LIN {X -0.182,Y -626.109,Z 300.159,A 0.000,B 0.000,C 90.000,E1 244.717} C_DIS
LIN {X -0.135,Y -624.501,Z 300.155,A 0.000,B 0.000,C 90.000,E1 243.948} C_DIS
LIN {X -0.103,Y -622.641,Z 300.151,A 0.000,B 0.000,C 90.000,E1 243.179} C_DIS
LIN {X -0.091,Y -619.995,Z 300.145,A 0.000,B 0.000,C 90.000,E1 242.153} C_DIS
LIN {X 0.159,Y -616.323,Z 300.138,A 0.000,B 0.000,C 90.000,E1 240.845} C_DIS
LIN {X -0.188,Y -612.551,Z 300.131,A 0.000,B 0.000,C 90.000,E1 239.587} C_DIS
LIN {X -0.081,Y -608.634,Z 300.124,A 0.000,B 0.000,C 90.000,E1 238.280} C_DIS
LIN {X 0.080,Y -604.709,Z 300.117,A 0.000,B 0.000,C 90.000,E1 236.962} C_DIS
LIN {X 0.094,Y -599.962,Z 300.108,A 0.000,B 0.000,C 90.000,E1 235.388} C_DIS
LIN {X -0.124,Y -596.687,Z 300.102,A 0.000,B 0.000,C 90.000,E1 234.356} C_DIS
LIN {X -0.079,Y -591.376,Z 300.093,A 0.000,B 0.000,C 90.000,E1 232.763} C_DIS
LIN {X -0.207,Y -584.502,Z 300.081,A 0.000,B 0.000,C 90.000,E1 230.642} C_DIS
LIN {X -0.209,Y -580.122,Z 300.074,A 0.000,B 0.000,C 90.000,E1 229.299} C_DIS
LIN {X 0.078,Y -573.427,Z 300.062,A 0.000,B 0.000,C 90.000,E1 227.106} C_DIS
LIN {X 0.222,Y -569.220,Z 300.054,A 0.000,B 0.000,C 90.000,E1 225.729} C_DIS
LIN {X -0.015,Y -564.128,Z 300.045,A 0.000,B 0.000,C 90.000,E1 224.109} C_DIS
LIN {X -0.037,Y -559.947,Z 300.037,A 0.000,B 0.000,C 90.000,E1 222.732} C_DIS
LIN {X -0.107,Y -555.813,Z 300.030,A 0.000,B 0.000,C 90.000,E1 221.353} C_DIS
LIN {X 0.230,Y -550.744,Z 300.020,A 0.000,B 0.000,C 90.000,E1 219.644} C_DIS
LIN {X -0.267,Y -544.758,Z 300.009,A 0.000,B 0.000,C 90.000,E1 217.729} C_DIS
LIN {X -0.126,Y -541.410,Z 300.003,A 0.000,B 0.000,C 90.000,E1 216.583} C_DIS
LIN {X 0.135,Y -534.785,Z 299.991,A 0.000,B 0.000,C 90.000,E1 214.278} C_DIS
LIN {X -0.097,Y -528.365,Z 299.978,A 0.000,B 0.000,C 90.000,E1 212.005} C_DIS
LIN {X -0.297,Y -523.035,Z 299.967,A 0.000,B 0.000,C 90.000,E1 210.001} C_DIS
LIN {X 0.222,Y -519.344,Z 299.958,A 0.000,B 0.000,C 90.000,E1 208.487} C_DIS
LIN {X -0.257,Y -514.359,Z 299.947,A 0.000,B 0.000,C 90.000,E1 206.488} C_DIS
LIN {X 0.058,Y -509.624,Z 299.936,A 0.000,B 0.000,C 90.000,E1 204.387} C_DIS
LIN {X -0.170,Y -505.196,Z 299.924,A 0.000,B 0.000,C 90.000,E1 202.333} C_DIS
LIN {X -0.150,Y -500.375,Z 299.911,A 0.000,B 0.000,C 90.000,E1 199.939} C_DIS
LIN {X -0.081,Y -495.359,Z 299.896,A 0.000,B 0.000,C 90.000,E1 197.221} C_DIS
LIN {X 0.007,Y -490.770,Z 299.880,A 0.000,B 0.000,C 90.000,E1 194.481} C_DIS
LIN {X 0.162,Y -488.457,Z 299.872,A 0.000,B 0.000,C 90.000,E1 192.939} C_DIS
LIN {X 0.166,Y -484.922,Z 299.858,A 0.000,B 0.000,C 90.000,E1 190.489} C_DIS
LIN {X -0.009,Y -481.708,Z 299.845,A 0.000,B 0.000,C 90.000,E1 188.049} C_DIS
LIN {X -0.052,Y -479.486,Z 299.834,A 0.000,B 0.000,C 90.000,E1 186.201} C_DIS
LIN {X -0.099,Y -476.814,Z 299.821,A 0.000,B 0.000,C 90.000,E1 183.726} C_DIS
LIN {X -0.082,Y -474.710,Z 299.809,A 0.000,B 0.000,C 90.000,E1 181.547} C_DIS
LIN {X 0.154,Y -472.452,Z 299.791,A 0.000,B 0.000,C 90.000,E1 178.396} C_DIS
LIN {X -0.120,Y -470.977,Z 299.774,A 0.000,B 0.000,C 90.000,E1 175.298} C_DIS
LIN {X -0.174,Y -470.415,Z 299.762,A 0.000,B 0.000,C 90.000,E1 173.109} C_DIS
LIN {X -0.218,Y -470.146,Z 299.753,A 0.000,B 0.000,C 90.000,E1 171.546} C_DIS
LIN {X -0.165,Y -470.044,Z 299.741,A 0.000,B 0.000,C 90.000,E1 169.342} C_DIS
LIN {X -0.162,Y -470.689,Z 299.720,A 0.000,B 0.000,C 90.000,E1 165.574} C_DIS
LIN {X 0.121,Y -471.798,Z 299.706,A 0.000,B 0.000,C 90.000,E1 163.032} C_DIS
LIN {X -0.060,Y -473.445,Z 299.692,A 0.000,B 0.000,C 90.000,E1 160.550} C_DIS
LIN {X 0.149,Y -475.397,Z 299.678,A 0.000,B 0.000,C 90.000,E1 158.028} C_DIS
LIN {X 0.148,Y -478.180,Z 299.663,A 0.000,B 0.000,C 90.000,E1 155.229} C_DIS
LIN {X 0.212,Y -481.326,Z 299.649,A 0.000,B 0.000,C 90.000,E1 152.743} C_DIS
LIN {X -0.264,Y -485.148,Z 299.635,A 0.000,B 0.000,C 90.000,E1 150.333} C_DIS
LIN {X -0.010,Y -487.281,Z 299.628,A 0.000,B 0.000,C 90.000,E1 149.076} C_DIS
LIN {X 0.181,Y -491.179,Z 299.616,A 0.000,B 0.000,C 90.000,E1 146.914} C_DIS
LIN {X 0.075,Y -494.680,Z 299.606,A 0.000,B 0.000,C 90.000,E1 145.102} C_DIS
LIN {X -0.221,Y -497.526,Z 299.598,A 0.000,B 0.000,C 90.000,E1 143.623} C_DIS
LIN {X -0.045,Y -499.723,Z 299.591,A 0.000,B 0.000,C 90.000,E1 142.396} C_DIS
LIN {X 0.044,Y -502.272,Z 299.583,A 0.000,B 0.000,C 90.000,E1 140.884} C_DIS
LIN {X 0.009,Y -503.703,Z 299.578,A 0.000,B 0.000,C 90.000,E1 139.989} C_DIS
LIN {X 0.206,Y -505.330,Z 299.571,A 0.000,B 0.000,C 90.000,E1 138.771} C_DIS
LIN {X -0.174,Y -506.358,Z 299.566,A 0.000,B 0.000,C 90.000,E1 137.919} C_DIS
LIN {X 0.174,Y -507.145,Z 299.561,A 0.000,B 0.000,C 90.000,E1 136.986} C_DIS
LIN {X -0.075,Y -507.587,Z 299.558,A 0.000,B 0.000,C 90.000,E1 136.419} C_DIS
LIN {X 0.284,Y -508.000,Z 299.553,A 0.000,B 0.000,C 90.000,E1 135.486} C_DIS
LIN {X -0.197,Y -508.143,Z 299.546,A 0.000,B 0.000,C 90.000,E1 134.352} C_DIS
LIN {X 0.037,Y -507.836,Z 299.540,A 0.000,B 0.000,C 90.000,E1 133.137} C_DIS
LIN {X 0.055,Y -507.294,Z 299.535,A 0.000,B 0.000,C 90.000,E1 132.243} C_DIS
LIN {X 0.031,Y -506.498,Z 299.530,A 0.000,B 0.000,C 90.000,E1 131.353} C_DIS
LIN {X 0.150,Y -504.769,Z 299.522,A 0.000,B 0.000,C 90.000,E1 129.850} C_DIS
LIN {X -0.197,Y -502.345,Z 299.512,A 0.000,B 0.000,C 90.000,E1 128.096} C_DIS
LIN {X 0.044,Y -500.568,Z 299.505,A 0.000,B 0.000,C 90.000,E1 126.870} C_DIS
LIN {X -0.039,Y -498.718,Z 299.498,A 0.000,B 0.000,C 90.000,E1 125.678} C_DIS
LIN {X -0.146,Y -496.550,Z 299.492,A 0.000,B 0.000,C 90.000,E1 124.485} C_DIS
LIN {X -0.021,Y -493.751,Z 299.483,A 0.000,B 0.000,C 90.000,E1 122.959} C_DIS
LIN {X -0.222,Y -490.785,Z 299.475,A 0.000,B 0.000,C 90.000,E1 121.465} C_DIS
LIN {X -0.066,Y -487.195,Z 299.465,A 0.000,B 0.000,C 90.000,E1 119.617} C_DIS
LIN {X 0.211,Y -484.805,Z 299.458,A 0.000,B 0.000,C 90.000,E1 118.359} C_DIS
LIN {X -0.021,Y -480.543,Z 299.446,A 0.000,B 0.000,C 90.000,E1 116.232} C_DIS
LIN {X -0.144,Y -476.269,Z 299.434,A 0.000,B 0.000,C 90.000,E1 114.079} C_DIS
LIN {X -0.141,Y -472.067,Z 299.422,A 0.000,B 0.000,C 90.000,E1 111.897} C_DIS
LIN {X -0.207,Y -467.442,Z 299.408,A 0.000,B 0.000,C 90.000,E1 109.396} C_DIS
LIN {X -0.204,Y -463.065,Z 299.394,A 0.000,B 0.000,C 90.000,E1 106.913} C_DIS
LIN {X 0.198,Y -463.061,Z 299.394,A 0.000,B 0.000,C 90.000,E1 106.858} C_DIS
LIN {X -0.082,Y -467.666,Z 299.383,A 0.000,B 0.000,C 90.000,E1 104.954} C_DIS
LIN {X -0.093,Y -473.980,Z 299.362,A 0.000,B 0.000,C 90.000,E1 101.186} C_DIS
LIN {X -0.125,Y -475.882,Z 299.357,A 0.000,B 0.000,C 90.000,E1 100.254} C_DIS
LIN {X 0.183,Y -476.341,Z 299.355,A 0.000,B 0.000,C 90.000,E1 99.905} C_DIS
LIN {X 0.140,Y -481.850,Z 299.331,A 0.000,B 0.000,C 90.000,E1 95.568} C_DIS
LIN {X -0.013,Y -482.187,Z 299.329,A 0.000,B 0.000,C 90.000,E1 95.277} C_DIS
LIN {X -0.079,Y -485.348,Z 299.305,A 0.000,B 0.000,C 90.000,E1 90.974} C_DIS
LIN {X 0.230,Y -485.533,Z 299.304,A 0.000,B 0.000,C 90.000,E1 90.630} C_DIS
LIN {X -0.047,Y -486.338,Z 299.282,A 0.000,B 0.000,C 90.000,E1 86.674} C_DIS
LIN {X 0.088,Y -486.278,Z 299.278,A 0.000,B 0.000,C 90.000,E1 86.045} C_DIS
LIN {X -0.193,Y -484.694,Z 299.254,A 0.000,B 0.000,C 90.000,E1 81.781} C_DIS
LIN {X 0.155,Y -484.553,Z 299.253,A 0.000,B 0.000,C 90.000,E1 81.432} C_DIS
LIN {X 0.024,Y -480.493,Z 299.227,A 0.000,B 0.000,C 90.000,E1 76.825} C_DIS
LIN {X 0.147,Y -474.643,Z 299.203,A 0.000,B 0.000,C 90.000,E1 72.543} C_DIS
LIN {X -0.098,Y -481.750,Z 299.187,A 0.000,B 0.000,C 90.000,E1 69.699} C_DIS
LIN {X -0.059,Y -487.505,Z 299.175,A 0.000,B 0.000,C 90.000,E1 67.539} C_DIS
LIN {X -0.122,Y -493.376,Z 299.163,A 0.000,B 0.000,C 90.000,E1 65.409} C_DIS
LIN {X 0.177,Y -499.347,Z 299.152,A 0.000,B 0.000,C 90.000,E1 63.256} C_DIS
LIN {X 0.100,Y -504.591,Z 299.142,A 0.000,B 0.000,C 90.000,E1 61.463} C_DIS
LIN {X -0.188,Y -510.675,Z 299.130,A 0.000,B 0.000,C 90.000,E1 59.410} C_DIS
LIN {X -0.053,Y -516.724,Z 299.118,A 0.000,B 0.000,C 90.000,E1 57.327} C_DIS
LIN {X -0.240,Y -520.932,Z 299.110,A 0.000,B 0.000,C 90.000,E1 55.881} C_DIS
LIN {X -0.012,Y -524.250,Z 299.104,A 0.000,B 0.000,C 90.000,E1 54.689} C_DIS
LIN {X 0.239,Y -528.043,Z 299.096,A 0.000,B 0.000,C 90.000,E1 53.210} C_DIS
LIN {X 0.166,Y -530.153,Z 299.091,A 0.000,B 0.000,C 90.000,E1 52.351} C_DIS
LIN {X -0.317,Y -532.828,Z 299.085,A 0.000,B 0.000,C 90.000,E1 51.251} C_DIS
LIN {X -0.017,Y -535.818,Z 299.077,A 0.000,B 0.000,C 90.000,E1 49.784} C_DIS
LIN {X -0.083,Y -537.922,Z 299.070,A 0.000,B 0.000,C 90.000,E1 48.647} C_DIS
LIN {X 0.243,Y -539.780,Z 299.064,A 0.000,B 0.000,C 90.000,E1 47.472} C_DIS
LIN {X 0.225,Y -540.990,Z 299.059,A 0.000,B 0.000,C 90.000,E1 46.620} C_DIS
LIN {X 0.210,Y -542.324,Z 299.053,A 0.000,B 0.000,C 90.000,E1 45.486} C_DIS
LIN {X -0.171,Y -543.078,Z 299.048,A 0.000,B 0.000,C 90.000,E1 44.676} C_DIS
LIN {X -0.157,Y -543.869,Z 299.042,A 0.000,B 0.000,C 90.000,E1 43.542} C_DIS
LIN {X -0.098,Y -544.655,Z 299.032,A 0.000,B 0.000,C 90.000,E1 41.838} C_DIS
LIN {X -0.032,Y -544.905,Z 299.026,A 0.000,B 0.000,C 90.000,E1 40.701} C_DIS
LIN {X 0.035,Y -544.893,Z 299.020,A 0.000,B 0.000,C 90.000,E1 39.564} C_DIS
LIN {X -0.282,Y -544.756,Z 299.015,A 0.000,B 0.000,C 90.000,E1 38.749} C_DIS
LIN {X -0.174,Y -544.378,Z 299.010,A 0.000,B 0.000,C 90.000,E1 37.890} C_DIS
LIN {X 0.005,Y -543.528,Z 299.003,A 0.000,B 0.000,C 90.000,E1 36.457} C_DIS
LIN {X 0.133,Y -542.653,Z 298.996,A 0.000,B 0.000,C 90.000,E1 35.311} C_DIS
LIN {X -0.044,Y -541.479,Z 298.988,A 0.000,B 0.000,C 90.000,E1 33.913} C_DIS
LIN {X 0.201,Y -540.148,Z 298.981,A 0.000,B 0.000,C 90.000,E1 32.467} C_DIS
LIN {X -0.148,Y -538.516,Z 298.971,A 0.000,B 0.000,C 90.000,E1 30.797} C_DIS
LIN {X -0.062,Y -536.827,Z 298.962,A 0.000,B 0.000,C 90.000,E1 29.077} C_DIS
LIN {X -0.080,Y -534.816,Z 298.950,A 0.000,B 0.000,C 90.000,E1 27.078} C_DIS
LIN {X -0.152,Y -532.853,Z 298.939,A 0.000,B 0.000,C 90.000,E1 25.079} C_DIS
LIN {X 0.131,Y -530.506,Z 298.925,A 0.000,B 0.000,C 90.000,E1 22.461} C_DIS
LIN {X 0.132,Y -528.251,Z 298.909,A 0.000,B 0.000,C 90.000,E1 19.577} C_DIS
LIN {X 0.020,Y -526.719,Z 298.896,A 0.000,B 0.000,C 90.000,E1 17.275} C_DIS
LIN {X 0.217,Y -525.316,Z 298.880,A 0.000,B 0.000,C 90.000,E1 14.356} C_DIS
LIN {X -0.064,Y -524.607,Z 298.869,A 0.000,B 0.000,C 90.000,E1 12.355} C_DIS
LIN {X 0.027,Y -524.180,Z 298.859,A 0.000,B 0.000,C 90.000,E1 10.602} C_DIS
LIN {X 0.028,Y -523.977,Z 298.848,A 0.000,B 0.000,C 90.000,E1 8.568} C_DIS
LIN {X -0.116,Y -524.085,Z 298.835,A 0.000,B 0.000,C 90.000,E1 6.258} C_DIS
LIN {X -0.217,Y -524.347,Z 298.827,A 0.000,B 0.000,C 90.000,E1 4.816} C_DIS
LIN {X 0.208,Y -524.558,Z 298.822,A 0.000,B 0.000,C 90.000,E1 3.898} C_DIS
LIN {X 0.074,Y -525.115,Z 298.815,A 0.000,B 0.000,C 90.000,E1 2.751} C_DIS
LIN {X -0.088,Y -525.738,Z 298.807,A 0.000,B 0.000,C 90.000,E1 1.318} C_DIS
LIN {X 0.015,Y -527.991,Z 298.788,A 0.000,B 0.000,C 90.000,E1 357.764} C_DIS
LIN {X -0.105,Y -529.771,Z 298.776,A 0.000,B 0.000,C 90.000,E1 355.755} C_DIS
LIN {X 0.151,Y -537.369,Z 298.744,A 0.000,B 0.000,C 90.000,E1 349.982} C_DIS
LIN {X 0.274,Y -546.360,Z 298.722,A 0.000,B 0.000,C 90.000,E1 345.992} C_DIS
LIN {X -0.070,Y -550.608,Z 298.713,A 0.000,B 0.000,C 90.000,E1 344.338} C_DIS
LIN {X 0.092,Y -555.900,Z 298.702,A 0.000,B 0.000,C 90.000,E1 342.362} C_DIS
LIN {X 0.033,Y -561.563,Z 298.691,A 0.000,B 0.000,C 90.000,E1 340.423} C_DIS
LIN {X -0.088,Y -568.480,Z 298.679,A 0.000,B 0.000,C 90.000,E1 338.230} C_DIS
LIN {X -0.154,Y -573.017,Z 298.671,A 0.000,B 0.000,C 90.000,E1 336.869} C_DIS
LIN {X -0.063,Y -578.480,Z 298.662,A 0.000,B 0.000,C 90.000,E1 335.229} C_DIS
LIN {X 0.019,Y -585.185,Z 298.652,A 0.000,B 0.000,C 90.000,E1 333.332} C_DIS
LIN {X 0.213,Y -589.950,Z 298.644,A 0.000,B 0.000,C 90.000,E1 331.975} C_DIS
LIN {X -0.028,Y -594.540,Z 298.637,A 0.000,B 0.000,C 90.000,E1 330.667} C_DIS
LIN {X 0.245,Y -600.852,Z 298.627,A 0.000,B 0.000,C 90.000,E1 328.791} C_DIS
LIN {X 0.368,Y -609.059,Z 298.614,A 0.000,B 0.000,C 90.000,E1 326.421} C_DIS
LIN {X -0.242,Y -616.568,Z 298.602,A 0.000,B 0.000,C 90.000,E1 324.402} C_DIS
LIN {X 0.137,Y -620.115,Z 298.596,A 0.000,B 0.000,C 90.000,E1 323.336} C_DIS
LIN {X 0.072,Y -623.435,Z 298.591,A 0.000,B 0.000,C 90.000,E1 322.316} C_DIS
LIN {X 0.003,Y -627.305,Z 298.584,A 0.000,B 0.000,C 90.000,E1 321.045} C_DIS
LIN {X -0.235,Y -631.904,Z 298.575,A 0.000,B 0.000,C 90.000,E1 319.542} C_DIS
LIN {X 0.147,Y -635.674,Z 298.568,A 0.000,B 0.000,C 90.000,E1 318.243} C_DIS
LIN {X 0.240,Y -642.093,Z 298.556,A 0.000,B 0.000,C 90.000,E1 315.972} C_DIS
LIN {X -0.207,Y -646.536,Z 298.547,A 0.000,B 0.000,C 90.000,E1 314.514} C_DIS
LIN {X -0.049,Y -649.984,Z 298.540,A 0.000,B 0.000,C 90.000,E1 313.257} C_DIS
LIN {X 0.170,Y -653.282,Z 298.533,A 0.000,B 0.000,C 90.000,E1 312.000} C_DIS
LIN {X 0.027,Y -655.124,Z 298.529,A 0.000,B 0.000,C 90.000,E1 311.272} C_DIS
LIN {X -0.082,Y -657.386,Z 298.524,A 0.000,B 0.000,C 90.000,E1 310.297} C_DIS
LIN {X 0.349,Y -659.514,Z 298.518,A 0.000,B 0.000,C 90.000,E1 309.277} C_DIS
LIN {X -0.147,Y -661.854,Z 298.512,A 0.000,B 0.000,C 90.000,E1 308.096} C_DIS
LIN {X 0.347,Y -663.452,Z 298.506,A 0.000,B 0.000,C 90.000,E1 307.076} C_DIS
LIN {X -0.030,Y -664.474,Z 298.502,A 0.000,B 0.000,C 90.000,E1 306.377} C_DIS
LIN {X -0.007,Y -665.299,Z 298.498,A 0.000,B 0.000,C 90.000,E1 305.644} C_DIS
LIN {X 0.061,Y -665.747,Z 298.495,A 0.000,B 0.000,C 90.000,E1 305.152} C_DIS
LIN {X 0.327,Y -666.190,Z 298.489,A 0.000,B 0.000,C 90.000,E1 303.913} C_DIS
LIN {X -0.026,Y -666.275,Z 298.485,A 0.000,B 0.000,C 90.000,E1 303.214} C_DIS
LIN {X 0.312,Y -665.993,Z 298.479,A 0.000,B 0.000,C 90.000,E1 302.212} C_DIS
LIN {X 0.026,Y -665.658,Z 298.476,A 0.000,B 0.000,C 90.000,E1 301.750} C_DIS
LIN {X 0.227,Y -664.792,Z 298.472,A 0.000,B 0.000,C 90.000,E1 301.003} C_DIS
LIN {X 0.078,Y -663.635,Z 298.468,A 0.000,B 0.000,C 90.000,E1 300.285} C_DIS
LIN {X -0.190,Y -661.626,Z 298.463,A 0.000,B 0.000,C 90.000,E1 299.333} C_DIS
LIN {X -0.236,Y -659.458,Z 298.457,A 0.000,B 0.000,C 90.000,E1 298.359} C_DIS
LIN {X -0.186,Y -656.523,Z 298.451,A 0.000,B 0.000,C 90.000,E1 297.129} C_DIS
LIN {X -0.192,Y -653.341,Z 298.444,A 0.000,B 0.000,C 90.000,E1 295.899} C_DIS
LIN {X -0.050,Y -650.744,Z 298.438,A 0.000,B 0.000,C 90.000,E1 294.899} C_DIS
LIN {X 0.156,Y -647.411,Z 298.431,A 0.000,B 0.000,C 90.000,E1 293.643} C_DIS
LIN {X 0.122,Y -643.343,Z 298.423,A 0.000,B 0.000,C 90.000,E1 292.153} C_DIS
LIN {X 0.003,Y -639.359,Z 298.415,A 0.000,B 0.000,C 90.000,E1 290.663} C_DIS
LIN {X 0.169,Y -635.540,Z 298.406,A 0.000,B 0.000,C 90.000,E1 289.141} C_DIS
LIN {X 0.083,Y -629.583,Z 298.392,A 0.000,B 0.000,C 90.000,E1 286.622} C_DIS
LIN {X 0.239,Y -624.337,Z 298.378,A 0.000,B 0.000,C 90.000,E1 284.064} C_DIS
LIN {X 0.299,Y -619.586,Z 298.363,A 0.000,B 0.000,C 90.000,E1 281.243} C_DIS
LIN {X -0.158,Y -616.056,Z 298.347,A 0.000,B 0.000,C 90.000,E1 278.454} C_DIS
LIN {X -0.290,Y -613.529,Z 298.331,A 0.000,B 0.000,C 90.000,E1 275.625} C_DIS
LIN {X -0.019,Y -612.132,Z 298.315,A 0.000,B 0.000,C 90.000,E1 272.751} C_DIS
LIN {X -0.136,Y -611.738,Z 298.304,A 0.000,B 0.000,C 90.000,E1 270.688} C_DIS
LIN {X -0.289,Y -612.009,Z 298.289,A 0.000,B 0.000,C 90.000,E1 268.108} C_DIS
LIN {X -0.093,Y -614.280,Z 298.268,A 0.000,B 0.000,C 90.000,E1 264.204} C_DIS
LIN {X -0.260,Y -616.461,Z 298.255,A 0.000,B 0.000,C 90.000,E1 261.894} C_DIS
LIN {X -0.129,Y -620.046,Z 298.239,A 0.000,B 0.000,C 90.000,E1 259.050} C_DIS
LIN {X -0.073,Y -623.099,Z 298.228,A 0.000,B 0.000,C 90.000,E1 256.992} C_DIS
LIN {X 0.084,Y -625.017,Z 298.221,A 0.000,B 0.000,C 90.000,E1 255.700} C_DIS
LIN {X 0.024,Y -626.507,Z 298.215,A 0.000,B 0.000,C 90.000,E1 254.685} C_DIS
LIN {X 0.018,Y -627.423,Z 298.211,A 0.000,B 0.000,C 90.000,E1 253.921} C_DIS
LIN {X -0.011,Y -628.337,Z 298.205,A 0.000,B 0.000,C 90.000,E1 252.906} C_DIS
LIN {X -0.241,Y -629.516,Z 298.197,A 0.000,B 0.000,C 90.000,E1 251.402} C_DIS
LIN {X 0.155,Y -629.873,Z 298.192,A 0.000,B 0.000,C 90.000,E1 250.604} C_DIS
LIN {X 0.355,Y -630.024,Z 298.187,A 0.000,B 0.000,C 90.000,E1 249.571} C_DIS
LIN {X -0.037,Y -629.773,Z 298.181,A 0.000,B 0.000,C 90.000,E1 248.592} C_DIS
LIN {X -0.236,Y -629.487,Z 298.178,A 0.000,B 0.000,C 90.000,E1 248.103} C_DIS
LIN {X 0.179,Y -628.629,Z 298.173,A 0.000,B 0.000,C 90.000,E1 247.050} C_DIS
LIN {X -0.015,Y -627.694,Z 298.168,A 0.000,B 0.000,C 90.000,E1 246.305} C_DIS
LIN {X -0.195,Y -625.621,Z 298.161,A 0.000,B 0.000,C 90.000,E1 245.049} C_DIS
LIN {X -0.159,Y -624.119,Z 298.157,A 0.000,B 0.000,C 90.000,E1 244.280} C_DIS
LIN {X -0.135,Y -622.359,Z 298.153,A 0.000,B 0.000,C 90.000,E1 243.512} C_DIS
LIN {X -0.136,Y -619.093,Z 298.146,A 0.000,B 0.000,C 90.000,E1 242.231} C_DIS
LIN {X 0.093,Y -615.474,Z 298.139,A 0.000,B 0.000,C 90.000,E1 240.923} C_DIS
LIN {X -0.272,Y -611.743,Z 298.131,A 0.000,B 0.000,C 90.000,E1 239.665} C_DIS
LIN {X 0.137,Y -607.865,Z 298.124,A 0.000,B 0.000,C 90.000,E1 238.329} C_DIS
LIN {X -0.039,Y -603.959,Z 298.117,A 0.000,B 0.000,C 90.000,E1 237.041} C_DIS
LIN {X 0.051,Y -599.975,Z 298.110,A 0.000,B 0.000,C 90.000,E1 235.722} C_DIS
LIN {X -0.160,Y -596.694,Z 298.104,A 0.000,B 0.000,C 90.000,E1 234.689} C_DIS
LIN {X -0.074,Y -593.204,Z 298.098,A 0.000,B 0.000,C 90.000,E1 233.623} C_DIS
LIN {X 0.111,Y -587.118,Z 298.088,A 0.000,B 0.000,C 90.000,E1 231.743} C_DIS
LIN {X -0.217,Y -582.880,Z 298.080,A 0.000,B 0.000,C 90.000,E1 230.436} C_DIS
LIN {X 0.153,Y -575.978,Z 298.068,A 0.000,B 0.000,C 90.000,E1 228.243} C_DIS
LIN {X 0.073,Y -571.039,Z 298.059,A 0.000,B 0.000,C 90.000,E1 226.620} C_DIS
LIN {X -0.129,Y -565.920,Z 298.050,A 0.000,B 0.000,C 90.000,E1 225.000} C_DIS
LIN {X -0.026,Y -560.892,Z 298.041,A 0.000,B 0.000,C 90.000,E1 223.338} C_DIS
LIN {X -0.034,Y -555.877,Z 298.032,A 0.000,B 0.000,C 90.000,E1 221.676} C_DIS
LIN {X -0.113,Y -550.777,Z 298.022,A 0.000,B 0.000,C 90.000,E1 220.011} C_DIS
LIN {X 0.073,Y -546.500,Z 298.014,A 0.000,B 0.000,C 90.000,E1 218.588} C_DIS
LIN {X 0.298,Y -541.470,Z 298.005,A 0.000,B 0.000,C 90.000,E1 216.870} C_DIS
LIN {X 0.115,Y -534.747,Z 297.992,A 0.000,B 0.000,C 90.000,E1 214.612} C_DIS
LIN {X 0.296,Y -527.505,Z 297.978,A 0.000,B 0.000,C 90.000,E1 212.005} C_DIS
LIN {X -0.326,Y -522.900,Z 297.968,A 0.000,B 0.000,C 90.000,E1 210.335} C_DIS
LIN {X 0.237,Y -517.730,Z 297.957,A 0.000,B 0.000,C 90.000,E1 208.231} C_DIS
LIN {X -0.280,Y -512.769,Z 297.946,A 0.000,B 0.000,C 90.000,E1 206.232} C_DIS
LIN {X -0.321,Y -508.749,Z 297.936,A 0.000,B 0.000,C 90.000,E1 204.463} C_DIS
LIN {X 0.101,Y -504.343,Z 297.924,A 0.000,B 0.000,C 90.000,E1 202.333} C_DIS
LIN {X 0.093,Y -499.541,Z 297.911,A 0.000,B 0.000,C 90.000,E1 199.939} C_DIS
LIN {X 0.131,Y -494.572,Z 297.896,A 0.000,B 0.000,C 90.000,E1 197.221} C_DIS
LIN {X 0.192,Y -490.013,Z 297.881,A 0.000,B 0.000,C 90.000,E1 194.481} C_DIS
LIN {X -0.252,Y -487.727,Z 297.872,A 0.000,B 0.000,C 90.000,E1 193.008} C_DIS
LIN {X -0.163,Y -484.250,Z 297.859,A 0.000,B 0.000,C 90.000,E1 190.546} C_DIS
LIN {X 0.118,Y -481.096,Z 297.845,A 0.000,B 0.000,C 90.000,E1 188.049} C_DIS
LIN {X -0.097,Y -478.583,Z 297.833,A 0.000,B 0.000,C 90.000,E1 185.910} C_DIS
LIN {X -0.210,Y -476.033,Z 297.819,A 0.000,B 0.000,C 90.000,E1 183.440} C_DIS
LIN {X -0.210,Y -473.997,Z 297.807,A 0.000,B 0.000,C 90.000,E1 181.260} C_DIS
LIN {X -0.033,Y -472.274,Z 297.793,A 0.000,B 0.000,C 90.000,E1 178.740} C_DIS
LIN {X 0.162,Y -470.725,Z 297.776,A 0.000,B 0.000,C 90.000,E1 175.584} C_DIS
LIN {X -0.130,Y -470.076,Z 297.762,A 0.000,B 0.000,C 90.000,E1 173.109} C_DIS
LIN {X 0.001,Y -469.874,Z 297.755,A 0.000,B 0.000,C 90.000,E1 171.837} C_DIS
LIN {X -0.137,Y -469.675,Z 297.741,A 0.000,B 0.000,C 90.000,E1 169.342} C_DIS
LIN {X -0.085,Y -470.203,Z 297.722,A 0.000,B 0.000,C 90.000,E1 165.880} C_DIS
LIN {X -0.145,Y -471.236,Z 297.708,A 0.000,B 0.000,C 90.000,E1 163.378} C_DIS
LIN {X -0.035,Y -472.778,Z 297.694,A 0.000,B 0.000,C 90.000,E1 160.859} C_DIS
LIN {X 0.237,Y -473.976,Z 297.685,A 0.000,B 0.000,C 90.000,E1 159.263} C_DIS
LIN {X 0.024,Y -476.139,Z 297.671,A 0.000,B 0.000,C 90.000,E1 156.794} C_DIS
LIN {X -0.199,Y -479.259,Z 297.656,A 0.000,B 0.000,C 90.000,E1 154.024} C_DIS
LIN {X 0.106,Y -484.121,Z 297.637,A 0.000,B 0.000,C 90.000,E1 150.589} C_DIS
LIN {X -0.087,Y -486.691,Z 297.628,A 0.000,B 0.000,C 90.000,E1 149.076} C_DIS
LIN {X 0.088,Y -490.536,Z 297.616,A 0.000,B 0.000,C 90.000,E1 146.914} C_DIS
LIN {X 0.117,Y -493.407,Z 297.608,A 0.000,B 0.000,C 90.000,E1 145.388} C_DIS
LIN {X -0.205,Y -496.206,Z 297.599,A 0.000,B 0.000,C 90.000,E1 143.909} C_DIS
LIN {X -0.049,Y -498.408,Z 297.593,A 0.000,B 0.000,C 90.000,E1 142.683} C_DIS
LIN {X 0.017,Y -500.971,Z 297.584,A 0.000,B 0.000,C 90.000,E1 141.170} C_DIS
LIN {X -0.151,Y -502.860,Z 297.578,A 0.000,B 0.000,C 90.000,E1 139.989} C_DIS
LIN {X 0.033,Y -504.484,Z 297.571,A 0.000,B 0.000,C 90.000,E1 138.771} C_DIS
LIN {X 0.136,Y -505.242,Z 297.568,A 0.000,B 0.000,C 90.000,E1 138.162} C_DIS
LIN {X -0.247,Y -506.101,Z 297.563,A 0.000,B 0.000,C 90.000,E1 137.310} C_DIS
LIN {X 0.094,Y -506.767,Z 297.558,A 0.000,B 0.000,C 90.000,E1 136.377} C_DIS
LIN {X 0.077,Y -507.162,Z 297.553,A 0.000,B 0.000,C 90.000,E1 135.486} C_DIS
LIN {X 0.301,Y -507.308,Z 297.546,A 0.000,B 0.000,C 90.000,E1 134.271} C_DIS
LIN {X -0.061,Y -507.139,Z 297.541,A 0.000,B 0.000,C 90.000,E1 133.419} C_DIS
LIN {X 0.153,Y -506.426,Z 297.535,A 0.000,B 0.000,C 90.000,E1 132.204} C_DIS
LIN {X 0.160,Y -505.647,Z 297.530,A 0.000,B 0.000,C 90.000,E1 131.310} C_DIS
LIN {X -0.219,Y -504.645,Z 297.525,A 0.000,B 0.000,C 90.000,E1 130.458} C_DIS
LIN {X -0.020,Y -503.134,Z 297.518,A 0.000,B 0.000,C 90.000,E1 129.241} C_DIS
LIN {X 0.108,Y -501.090,Z 297.510,A 0.000,B 0.000,C 90.000,E1 127.729} C_DIS
LIN {X 0.075,Y -498.355,Z 297.500,A 0.000,B 0.000,C 90.000,E1 125.931} C_DIS
LIN {X 0.089,Y -496.811,Z 297.495,A 0.000,B 0.000,C 90.000,E1 125.025} C_DIS
LIN {X 0.066,Y -493.432,Z 297.485,A 0.000,B 0.000,C 90.000,E1 123.214} C_DIS
LIN {X 0.014,Y -491.122,Z 297.478,A 0.000,B 0.000,C 90.000,E1 122.005} C_DIS
LIN {X 0.178,Y -488.142,Z 297.469,A 0.000,B 0.000,C 90.000,E1 120.463} C_DIS
LIN {X 0.040,Y -485.166,Z 297.461,A 0.000,B 0.000,C 90.000,E1 118.949} C_DIS
LIN {X 0.052,Y -482.748,Z 297.454,A 0.000,B 0.000,C 90.000,E1 117.719} C_DIS
LIN {X 0.216,Y -479.099,Z 297.444,A 0.000,B 0.000,C 90.000,E1 115.848} C_DIS
LIN {X -0.119,Y -475.443,Z 297.433,A 0.000,B 0.000,C 90.000,E1 114.027} C_DIS
LIN {X -0.132,Y -471.269,Z 297.421,A 0.000,B 0.000,C 90.000,E1 111.844} C_DIS
LIN {X -0.059,Y -466.674,Z 297.407,A 0.000,B 0.000,C 90.000,E1 109.322} C_DIS
LIN {X 0.031,Y -462.724,Z 297.395,A 0.000,B 0.000,C 90.000,E1 107.040} C_DIS
LIN {X -0.010,Y -462.719,Z 297.395,A 0.000,B 0.000,C 90.000,E1 107.040} C_DIS
LIN {X -0.099,Y -467.796,Z 297.383,A 0.000,B 0.000,C 90.000,E1 104.898} C_DIS
LIN {X -0.128,Y -476.002,Z 297.357,A 0.000,B 0.000,C 90.000,E1 100.197} C_DIS
LIN {X -0.137,Y -477.010,Z 297.351,A 0.000,B 0.000,C 90.000,E1 99.265} C_DIS
LIN {X 0.146,Y -481.941,Z 297.331,A 0.000,B 0.000,C 90.000,E1 95.511} C_DIS
LIN {X -0.007,Y -482.210,Z 297.329,A 0.000,B 0.000,C 90.000,E1 95.220} C_DIS
LIN {X -0.068,Y -485.408,Z 297.305,A 0.000,B 0.000,C 90.000,E1 90.917} C_DIS
LIN {X 0.242,Y -485.528,Z 297.303,A 0.000,B 0.000,C 90.000,E1 90.573} C_DIS
LIN {X -0.036,Y -486.367,Z 297.281,A 0.000,B 0.000,C 90.000,E1 86.617} C_DIS
LIN {X -0.210,Y -486.367,Z 297.280,A 0.000,B 0.000,C 90.000,E1 86.331} C_DIS
LIN {X 0.124,Y -485.673,Z 297.273,A 0.000,B 0.000,C 90.000,E1 85.065} C_DIS
LIN {X -0.188,Y -484.691,Z 297.254,A 0.000,B 0.000,C 90.000,E1 81.724} C_DIS
LIN {X 0.160,Y -484.485,Z 297.252,A 0.000,B 0.000,C 90.000,E1 81.376} C_DIS
LIN {X 0.163,Y -480.661,Z 297.228,A 0.000,B 0.000,C 90.000,E1 77.061} C_DIS
LIN {X 0.129,Y -480.411,Z 297.227,A 0.000,B 0.000,C 90.000,E1 76.756} C_DIS
LIN {X -0.113,Y -474.423,Z 297.202,A 0.000,B 0.000,C 90.000,E1 72.362} C_DIS
LIN {X 0.048,Y -479.524,Z 297.190,A 0.000,B 0.000,C 90.000,E1 70.242} C_DIS
LIN {X -0.145,Y -485.198,Z 297.178,A 0.000,B 0.000,C 90.000,E1 68.103} C_DIS
LIN {X 0.123,Y -489.376,Z 297.170,A 0.000,B 0.000,C 90.000,E1 66.538} C_DIS
LIN {X -0.178,Y -493.591,Z 297.161,A 0.000,B 0.000,C 90.000,E1 65.049} C_DIS
LIN {X 0.013,Y -497.858,Z 297.153,A 0.000,B 0.000,C 90.000,E1 63.512} C_DIS
LIN {X 0.202,Y -503.972,Z 297.141,A 0.000,B 0.000,C 90.000,E1 61.385} C_DIS
LIN {X -0.092,Y -510.039,Z 297.130,A 0.000,B 0.000,C 90.000,E1 59.331} C_DIS
LIN {X -0.237,Y -514.395,Z 297.121,A 0.000,B 0.000,C 90.000,E1 57.867} C_DIS
LIN {X -0.035,Y -518.670,Z 297.113,A 0.000,B 0.000,C 90.000,E1 56.373} C_DIS
LIN {X 0.108,Y -522.812,Z 297.105,A 0.000,B 0.000,C 90.000,E1 54.895} C_DIS
LIN {X -0.088,Y -526.680,Z 297.097,A 0.000,B 0.000,C 90.000,E1 53.463} C_DIS
LIN {X 0.226,Y -529.520,Z 297.091,A 0.000,B 0.000,C 90.000,E1 52.271} C_DIS
LIN {X -0.264,Y -532.181,Z 297.084,A 0.000,B 0.000,C 90.000,E1 51.170} C_DIS
LIN {X 0.032,Y -534.577,Z 297.078,A 0.000,B 0.000,C 90.000,E1 49.989} C_DIS
LIN {X -0.046,Y -536.758,Z 297.071,A 0.000,B 0.000,C 90.000,E1 48.852} C_DIS
LIN {X -0.095,Y -538.647,Z 297.065,A 0.000,B 0.000,C 90.000,E1 47.715} C_DIS
LIN {X -0.125,Y -539.901,Z 297.060,A 0.000,B 0.000,C 90.000,E1 46.863} C_DIS
LIN {X -0.160,Y -541.317,Z 297.054,A 0.000,B 0.000,C 90.000,E1 45.729} C_DIS
LIN {X -0.169,Y -542.321,Z 297.048,A 0.000,B 0.000,C 90.000,E1 44.595} C_DIS
LIN {X -0.166,Y -543.093,Z 297.041,A 0.000,B 0.000,C 90.000,E1 43.461} C_DIS
LIN {X -0.125,Y -543.879,Z 297.032,A 0.000,B 0.000,C 90.000,E1 41.757} C_DIS
LIN {X -0.072,Y -544.051,Z 297.026,A 0.000,B 0.000,C 90.000,E1 40.620} C_DIS
LIN {X -0.049,Y -544.039,Z 297.021,A 0.000,B 0.000,C 90.000,E1 39.769} C_DIS
LIN {X 0.045,Y -543.894,Z 297.016,A 0.000,B 0.000,C 90.000,E1 38.910} C_DIS
LIN {X -0.282,Y -543.593,Z 297.012,A 0.000,B 0.000,C 90.000,E1 38.096} C_DIS
LIN {X -0.120,Y -542.787,Z 297.004,A 0.000,B 0.000,C 90.000,E1 36.664} C_DIS
LIN {X -0.004,Y -541.943,Z 296.997,A 0.000,B 0.000,C 90.000,E1 35.518} C_DIS
LIN {X -0.174,Y -540.545,Z 296.988,A 0.000,B 0.000,C 90.000,E1 33.833} C_DIS
LIN {X -0.231,Y -538.910,Z 296.978,A 0.000,B 0.000,C 90.000,E1 32.133} C_DIS
LIN {X 0.139,Y -537.525,Z 296.971,A 0.000,B 0.000,C 90.000,E1 30.669} C_DIS
LIN {X 0.203,Y -535.798,Z 296.961,A 0.000,B 0.000,C 90.000,E1 28.949} C_DIS
LIN {X -0.033,Y -534.093,Z 296.951,A 0.000,B 0.000,C 90.000,E1 27.257} C_DIS
LIN {X 0.059,Y -531.767,Z 296.939,A 0.000,B 0.000,C 90.000,E1 24.951} C_DIS
LIN {X -0.186,Y -529.403,Z 296.924,A 0.000,B 0.000,C 90.000,E1 22.386} C_DIS
LIN {X -0.091,Y -527.679,Z 296.913,A 0.000,B 0.000,C 90.000,E1 20.355} C_DIS
LIN {X -0.240,Y -526.899,Z 296.907,A 0.000,B 0.000,C 90.000,E1 19.214} C_DIS
LIN {X -0.050,Y -525.565,Z 296.895,A 0.000,B 0.000,C 90.000,E1 17.166} C_DIS
LIN {X 0.120,Y -524.139,Z 296.879,A 0.000,B 0.000,C 90.000,E1 14.245} C_DIS
LIN {X -0.182,Y -523.401,Z 296.868,A 0.000,B 0.000,C 90.000,E1 12.243} C_DIS
LIN {X -0.101,Y -522.902,Z 296.857,A 0.000,B 0.000,C 90.000,E1 10.197} C_DIS
LIN {X -0.131,Y -522.737,Z 296.845,A 0.000,B 0.000,C 90.000,E1 8.163} C_DIS
LIN {X 0.152,Y -522.951,Z 296.831,A 0.000,B 0.000,C 90.000,E1 5.511} C_DIS
LIN {X -0.171,Y -523.827,Z 296.815,A 0.000,B 0.000,C 90.000,E1 2.636} C_DIS
LIN {X 0.131,Y -524.569,Z 296.805,A 0.000,B 0.000,C 90.000,E1 0.859} C_DIS
LIN {X -0.020,Y -526.647,Z 296.788,A 0.000,B 0.000,C 90.000,E1 357.764} C_DIS
LIN {X -0.174,Y -528.396,Z 296.776,A 0.000,B 0.000,C 90.000,E1 355.755} C_DIS
LIN {X -0.072,Y -535.561,Z 296.746,A 0.000,B 0.000,C 90.000,E1 350.274} C_DIS
LIN {X -0.246,Y -538.893,Z 296.736,A 0.000,B 0.000,C 90.000,E1 348.578} C_DIS
LIN {X 0.031,Y -545.005,Z 296.722,A 0.000,B 0.000,C 90.000,E1 345.992} C_DIS
LIN {X 0.186,Y -549.258,Z 296.713,A 0.000,B 0.000,C 90.000,E1 344.283} C_DIS
LIN {X 0.058,Y -555.342,Z 296.700,A 0.000,B 0.000,C 90.000,E1 342.054} C_DIS
LIN {X 0.108,Y -561.900,Z 296.688,A 0.000,B 0.000,C 90.000,E1 339.826} C_DIS
LIN {X 0.260,Y -567.168,Z 296.679,A 0.000,B 0.000,C 90.000,E1 338.156} C_DIS
LIN {X 0.181,Y -571.747,Z 296.671,A 0.000,B 0.000,C 90.000,E1 336.794} C_DIS
LIN {X -0.287,Y -579.148,Z 296.659,A 0.000,B 0.000,C 90.000,E1 334.665} C_DIS
LIN {X 0.192,Y -584.949,Z 296.650,A 0.000,B 0.000,C 90.000,E1 332.999} C_DIS
LIN {X -0.130,Y -589.632,Z 296.643,A 0.000,B 0.000,C 90.000,E1 331.691} C_DIS
LIN {X 0.146,Y -594.209,Z 296.635,A 0.000,B 0.000,C 90.000,E1 330.333} C_DIS
LIN {X 0.189,Y -599.601,Z 296.626,A 0.000,B 0.000,C 90.000,E1 328.742} C_DIS
LIN {X 0.332,Y -606.884,Z 296.615,A 0.000,B 0.000,C 90.000,E1 326.628} C_DIS
LIN {X 0.166,Y -614.448,Z 296.603,A 0.000,B 0.000,C 90.000,E1 324.562} C_DIS
LIN {X 0.015,Y -618.096,Z 296.598,A 0.000,B 0.000,C 90.000,E1 323.543} C_DIS
LIN {X 0.039,Y -621.497,Z 296.592,A 0.000,B 0.000,C 90.000,E1 322.512} C_DIS
LIN {X -0.171,Y -625.493,Z 296.585,A 0.000,B 0.000,C 90.000,E1 321.251} C_DIS
LIN {X 0.040,Y -630.133,Z 296.576,A 0.000,B 0.000,C 90.000,E1 319.703} C_DIS
LIN {X -0.086,Y -633.912,Z 296.569,A 0.000,B 0.000,C 90.000,E1 318.447} C_DIS
LIN {X 0.145,Y -638.911,Z 296.559,A 0.000,B 0.000,C 90.000,E1 316.662} C_DIS
LIN {X 0.100,Y -643.283,Z 296.551,A 0.000,B 0.000,C 90.000,E1 315.162} C_DIS
LIN {X -0.192,Y -646.205,Z 296.545,A 0.000,B 0.000,C 90.000,E1 314.190} C_DIS
LIN {X 0.019,Y -648.957,Z 296.540,A 0.000,B 0.000,C 90.000,E1 313.176} C_DIS
LIN {X 0.220,Y -652.254,Z 296.533,A 0.000,B 0.000,C 90.000,E1 311.919} C_DIS
LIN {X 0.081,Y -654.644,Z 296.528,A 0.000,B 0.000,C 90.000,E1 310.943} C_DIS
LIN {X -0.022,Y -656.892,Z 296.522,A 0.000,B 0.000,C 90.000,E1 309.967} C_DIS
LIN {X -0.099,Y -658.910,Z 296.517,A 0.000,B 0.000,C 90.000,E1 308.991} C_DIS
LIN {X -0.158,Y -660.714,Z 296.511,A 0.000,B 0.000,C 90.000,E1 308.016} C_DIS
LIN {X -0.166,Y -661.916,Z 296.507,A 0.000,B 0.000,C 90.000,E1 307.282} C_DIS
LIN {X -0.071,Y -663.294,Z 296.502,A 0.000,B 0.000,C 90.000,E1 306.297} C_DIS
LIN {X 0.046,Y -664.319,Z 296.496,A 0.000,B 0.000,C 90.000,E1 305.311} C_DIS
LIN {X 0.174,Y -664.716,Z 296.491,A 0.000,B 0.000,C 90.000,E1 304.326} C_DIS
LIN {X -0.066,Y -664.937,Z 296.485,A 0.000,B 0.000,C 90.000,E1 303.372} C_DIS
LIN {X -0.300,Y -664.713,Z 296.480,A 0.000,B 0.000,C 90.000,E1 302.418} C_DIS
LIN {X -0.243,Y -664.428,Z 296.477,A 0.000,B 0.000,C 90.000,E1 301.926} C_DIS
LIN {X -0.060,Y -663.627,Z 296.473,A 0.000,B 0.000,C 90.000,E1 301.180} C_DIS
LIN {X -0.226,Y -662.518,Z 296.469,A 0.000,B 0.000,C 90.000,E1 300.463} C_DIS
LIN {X -0.068,Y -661.097,Z 296.465,A 0.000,B 0.000,C 90.000,E1 299.716} C_DIS
LIN {X 0.000,Y -658.416,Z 296.458,A 0.000,B 0.000,C 90.000,E1 298.487} C_DIS
LIN {X 0.031,Y -655.475,Z 296.451,A 0.000,B 0.000,C 90.000,E1 297.257} C_DIS
LIN {X -0.099,Y -652.976,Z 296.446,A 0.000,B 0.000,C 90.000,E1 296.283} C_DIS
LIN {X 0.136,Y -649.725,Z 296.439,A 0.000,B 0.000,C 90.000,E1 295.027} C_DIS
LIN {X -0.268,Y -646.373,Z 296.432,A 0.000,B 0.000,C 90.000,E1 293.823} C_DIS
LIN {X 0.335,Y -641.619,Z 296.423,A 0.000,B 0.000,C 90.000,E1 292.025} C_DIS
LIN {X -0.047,Y -637.684,Z 296.414,A 0.000,B 0.000,C 90.000,E1 290.556} C_DIS
LIN {X 0.116,Y -633.248,Z 296.404,A 0.000,B 0.000,C 90.000,E1 288.779} C_DIS
LIN {X 0.170,Y -628.488,Z 296.393,A 0.000,B 0.000,C 90.000,E1 286.749} C_DIS
LIN {X -0.095,Y -623.718,Z 296.380,A 0.000,B 0.000,C 90.000,E1 284.481} C_DIS
LIN {X -0.271,Y -618.454,Z 296.363,A 0.000,B 0.000,C 90.000,E1 281.422} C_DIS
LIN {X -0.171,Y -615.407,Z 296.350,A 0.000,B 0.000,C 90.000,E1 279.095} C_DIS
LIN {X 0.094,Y -612.502,Z 296.333,A 0.000,B 0.000,C 90.000,E1 275.967} C_DIS
LIN {X -0.018,Y -610.861,Z 296.316,A 0.000,B 0.000,C 90.000,E1 272.865} C_DIS
LIN {X 0.112,Y -610.409,Z 296.303,A 0.000,B 0.000,C 90.000,E1 270.516} C_DIS
LIN {X 0.223,Y -610.677,Z 296.290,A 0.000,B 0.000,C 90.000,E1 268.167} C_DIS
LIN {X 0.095,Y -612.688,Z 296.270,A 0.000,B 0.000,C 90.000,E1 264.546} C_DIS
LIN {X 0.170,Y -615.108,Z 296.255,A 0.000,B 0.000,C 90.000,E1 261.951} C_DIS
LIN {X 0.257,Y -618.704,Z 296.240,A 0.000,B 0.000,C 90.000,E1 259.106} C_DIS
LIN {X 0.145,Y -621.749,Z 296.228,A 0.000,B 0.000,C 90.000,E1 257.061} C_DIS
LIN {X 0.210,Y -624.067,Z 296.220,A 0.000,B 0.000,C 90.000,E1 255.519} C_DIS
LIN {X -0.026,Y -625.542,Z 296.214,A 0.000,B 0.000,C 90.000,E1 254.519} C_DIS
LIN {X 0.126,Y -626.434,Z 296.210,A 0.000,B 0.000,C 90.000,E1 253.740} C_DIS
LIN {X -0.121,Y -627.519,Z 296.203,A 0.000,B 0.000,C 90.000,E1 252.489} C_DIS
LIN {X -0.166,Y -628.448,Z 296.196,A 0.000,B 0.000,C 90.000,E1 251.221} C_DIS
LIN {X 0.220,Y -628.758,Z 296.191,A 0.000,B 0.000,C 90.000,E1 250.423} C_DIS
LIN {X -0.186,Y -628.847,Z 296.186,A 0.000,B 0.000,C 90.000,E1 249.444} C_DIS
LIN {X -0.006,Y -628.518,Z 296.180,A 0.000,B 0.000,C 90.000,E1 248.411} C_DIS
LIN {X -0.184,Y -627.762,Z 296.174,A 0.000,B 0.000,C 90.000,E1 247.411} C_DIS
LIN {X 0.193,Y -626.931,Z 296.170,A 0.000,B 0.000,C 90.000,E1 246.613} C_DIS
LIN {X -0.007,Y -625.434,Z 296.165,A 0.000,B 0.000,C 90.000,E1 245.613} C_DIS
LIN {X 0.027,Y -624.121,Z 296.160,A 0.000,B 0.000,C 90.000,E1 244.845} C_DIS
LIN {X 0.052,Y -622.557,Z 296.156,A 0.000,B 0.000,C 90.000,E1 244.076} C_DIS
LIN {X 0.063,Y -620.759,Z 296.152,A 0.000,B 0.000,C 90.000,E1 243.307} C_DIS
LIN {X 0.057,Y -618.822,Z 296.148,A 0.000,B 0.000,C 90.000,E1 242.538} C_DIS
LIN {X 0.011,Y -616.058,Z 296.142,A 0.000,B 0.000,C 90.000,E1 241.513} C_DIS
LIN {X 0.187,Y -612.407,Z 296.135,A 0.000,B 0.000,C 90.000,E1 240.205} C_DIS
LIN {X -0.187,Y -609.370,Z 296.129,A 0.000,B 0.000,C 90.000,E1 239.203} C_DIS
LIN {X 0.239,Y -606.290,Z 296.123,A 0.000,B 0.000,C 90.000,E1 238.122} C_DIS
LIN {X -0.044,Y -601.570,Z 296.114,A 0.000,B 0.000,C 90.000,E1 236.580} C_DIS
LIN {X 0.100,Y -598.352,Z 296.109,A 0.000,B 0.000,C 90.000,E1 235.515} C_DIS
LIN {X -0.135,Y -595.014,Z 296.103,A 0.000,B 0.000,C 90.000,E1 234.482} C_DIS
LIN {X 0.352,Y -589.717,Z 296.094,A 0.000,B 0.000,C 90.000,E1 232.844} C_DIS
LIN {X 0.256,Y -584.628,Z 296.085,A 0.000,B 0.000,C 90.000,E1 231.251} C_DIS
LIN {X 0.077,Y -581.231,Z 296.079,A 0.000,B 0.000,C 90.000,E1 230.194} C_DIS
LIN {X 0.020,Y -574.387,Z 296.067,A 0.000,B 0.000,C 90.000,E1 228.038} C_DIS
LIN {X 0.292,Y -569.440,Z 296.058,A 0.000,B 0.000,C 90.000,E1 226.377} C_DIS
LIN {X -0.258,Y -563.489,Z 296.047,A 0.000,B 0.000,C 90.000,E1 224.514} C_DIS
LIN {X 0.246,Y -557.602,Z 296.036,A 0.000,B 0.000,C 90.000,E1 222.528} C_DIS
LIN {X 0.140,Y -553.383,Z 296.029,A 0.000,B 0.000,C 90.000,E1 221.148} C_DIS
LIN {X 0.322,Y -549.976,Z 296.023,A 0.000,B 0.000,C 90.000,E1 220.011} C_DIS
LIN {X -0.235,Y -544.843,Z 296.013,A 0.000,B 0.000,C 90.000,E1 218.382} C_DIS
LIN {X -0.092,Y -541.471,Z 296.007,A 0.000,B 0.000,C 90.000,E1 217.237} C_DIS
LIN {X 0.037,Y -535.537,Z 295.996,A 0.000,B 0.000,C 90.000,E1 215.231} C_DIS
LIN {X 0.173,Y -532.233,Z 295.989,A 0.000,B 0.000,C 90.000,E1 214.072} C_DIS
LIN {X -0.041,Y -524.320,Z 295.973,A 0.000,B 0.000,C 90.000,E1 211.209} C_DIS
LIN {X 0.031,Y -518.280,Z 295.960,A 0.000,B 0.000,C 90.000,E1 208.871} C_DIS
LIN {X -0.133,Y -513.948,Z 295.951,A 0.000,B 0.000,C 90.000,E1 207.129} C_DIS
LIN {X -0.185,Y -508.528,Z 295.938,A 0.000,B 0.000,C 90.000,E1 204.771} C_DIS
LIN {X -0.151,Y -503.476,Z 295.924,A 0.000,B 0.000,C 90.000,E1 202.386} C_DIS
LIN {X -0.191,Y -498.668,Z 295.911,A 0.000,B 0.000,C 90.000,E1 199.993} C_DIS
LIN {X -0.186,Y -493.749,Z 295.896,A 0.000,B 0.000,C 90.000,E1 197.275} C_DIS
LIN {X -0.155,Y -489.262,Z 295.881,A 0.000,B 0.000,C 90.000,E1 194.537} C_DIS
LIN {X -0.140,Y -486.986,Z 295.872,A 0.000,B 0.000,C 90.000,E1 193.008} C_DIS
LIN {X 0.056,Y -483.984,Z 295.860,A 0.000,B 0.000,C 90.000,E1 190.838} C_DIS
LIN {X -0.145,Y -480.857,Z 295.847,A 0.000,B 0.000,C 90.000,E1 188.398} C_DIS
LIN {X -0.043,Y -478.055,Z 295.833,A 0.000,B 0.000,C 90.000,E1 185.910} C_DIS
LIN {X -0.172,Y -475.533,Z 295.819,A 0.000,B 0.000,C 90.000,E1 183.440} C_DIS
LIN {X -0.185,Y -473.547,Z 295.807,A 0.000,B 0.000,C 90.000,E1 181.260} C_DIS
LIN {X -0.021,Y -471.847,Z 295.793,A 0.000,B 0.000,C 90.000,E1 178.740} C_DIS
LIN {X -0.080,Y -470.449,Z 295.777,A 0.000,B 0.000,C 90.000,E1 175.927} C_DIS
LIN {X -0.147,Y -469.683,Z 295.762,A 0.000,B 0.000,C 90.000,E1 173.109} C_DIS
LIN {X -0.021,Y -469.481,Z 295.755,A 0.000,B 0.000,C 90.000,E1 171.837} C_DIS
LIN {X -0.171,Y -469.266,Z 295.741,A 0.000,B 0.000,C 90.000,E1 169.342} C_DIS
LIN {X 0.229,Y -469.614,Z 295.725,A 0.000,B 0.000,C 90.000,E1 166.464} C_DIS
LIN {X -0.209,Y -470.811,Z 295.708,A 0.000,B 0.000,C 90.000,E1 163.378} C_DIS
LIN {X -0.152,Y -472.577,Z 295.692,A 0.000,B 0.000,C 90.000,E1 160.550} C_DIS
LIN {X 0.088,Y -474.038,Z 295.681,A 0.000,B 0.000,C 90.000,E1 158.646} C_DIS
LIN {X -0.126,Y -476.320,Z 295.668,A 0.000,B 0.000,C 90.000,E1 156.177} C_DIS
LIN {X 0.116,Y -478.772,Z 295.656,A 0.000,B 0.000,C 90.000,E1 153.973} C_DIS
LIN {X -0.031,Y -483.619,Z 295.637,A 0.000,B 0.000,C 90.000,E1 150.589} C_DIS
LIN {X 0.203,Y -485.622,Z 295.630,A 0.000,B 0.000,C 90.000,E1 149.331} C_DIS
LIN {X 0.092,Y -489.377,Z 295.618,A 0.000,B 0.000,C 90.000,E1 147.199} C_DIS
LIN {X 0.095,Y -492.181,Z 295.609,A 0.000,B 0.000,C 90.000,E1 145.674} C_DIS
LIN {X 0.005,Y -495.461,Z 295.599,A 0.000,B 0.000,C 90.000,E1 143.863} C_DIS
LIN {X 0.144,Y -497.623,Z 295.593,A 0.000,B 0.000,C 90.000,E1 142.637} C_DIS
LIN {X -0.201,Y -500.181,Z 295.584,A 0.000,B 0.000,C 90.000,E1 141.170} C_DIS
LIN {X -0.259,Y -501.593,Z 295.579,A 0.000,B 0.000,C 90.000,E1 140.275} C_DIS
LIN {X -0.211,Y -503.648,Z 295.571,A 0.000,B 0.000,C 90.000,E1 138.771} C_DIS
LIN {X -0.115,Y -504.425,Z 295.568,A 0.000,B 0.000,C 90.000,E1 138.162} C_DIS
LIN {X 0.207,Y -505.284,Z 295.563,A 0.000,B 0.000,C 90.000,E1 137.229} C_DIS
LIN {X -0.176,Y -505.947,Z 295.558,A 0.000,B 0.000,C 90.000,E1 136.377} C_DIS
LIN {X 0.028,Y -506.371,Z 295.551,A 0.000,B 0.000,C 90.000,E1 135.162} C_DIS
LIN {X 0.008,Y -506.457,Z 295.546,A 0.000,B 0.000,C 90.000,E1 134.271} C_DIS
LIN {X -0.014,Y -506.283,Z 295.541,A 0.000,B 0.000,C 90.000,E1 133.380} C_DIS
LIN {X -0.160,Y -505.553,Z 295.534,A 0.000,B 0.000,C 90.000,E1 132.204} C_DIS
LIN {X -0.163,Y -504.788,Z 295.529,A 0.000,B 0.000,C 90.000,E1 131.310} C_DIS
LIN {X 0.160,Y -503.802,Z 295.524,A 0.000,B 0.000,C 90.000,E1 130.378} C_DIS
LIN {X 0.026,Y -502.294,Z 295.518,A 0.000,B 0.000,C 90.000,E1 129.197} C_DIS
LIN {X -0.250,Y -500.249,Z 295.509,A 0.000,B 0.000,C 90.000,E1 127.729} C_DIS
LIN {X -0.171,Y -497.945,Z 295.501,A 0.000,B 0.000,C 90.000,E1 126.217} C_DIS
LIN {X -0.159,Y -496.489,Z 295.496,A 0.000,B 0.000,C 90.000,E1 125.311} C_DIS
LIN {X -0.036,Y -493.679,Z 295.488,A 0.000,B 0.000,C 90.000,E1 123.785} C_DIS
LIN {X 0.026,Y -490.849,Z 295.479,A 0.000,B 0.000,C 90.000,E1 122.260} C_DIS
LIN {X -0.247,Y -487.274,Z 295.469,A 0.000,B 0.000,C 90.000,E1 120.463} C_DIS
LIN {X 0.026,Y -484.288,Z 295.461,A 0.000,B 0.000,C 90.000,E1 118.899} C_DIS
LIN {X -0.184,Y -481.253,Z 295.452,A 0.000,B 0.000,C 90.000,E1 117.385} C_DIS
LIN {X -0.061,Y -477.642,Z 295.442,A 0.000,B 0.000,C 90.000,E1 115.515} C_DIS
LIN {X 0.026,Y -474.600,Z 295.433,A 0.000,B 0.000,C 90.000,E1 113.951} C_DIS
LIN {X 0.021,Y -471.046,Z 295.423,A 0.000,B 0.000,C 90.000,E1 112.078} C_DIS
LIN {X 0.187,Y -467.505,Z 295.412,A 0.000,B 0.000,C 90.000,E1 110.174} C_DIS
LIN {X 0.178,Y -464.757,Z 295.404,A 0.000,B 0.000,C 90.000,E1 108.598} C_DIS
LIN {X -0.167,Y -462.388,Z 295.396,A 0.000,B 0.000,C 90.000,E1 107.221} C_DIS
LIN {X -0.207,Y -462.379,Z 295.396,A 0.000,B 0.000,C 90.000,E1 107.221} C_DIS
LIN {X -0.070,Y -467.914,Z 295.382,A 0.000,B 0.000,C 90.000,E1 104.828} C_DIS
LIN {X -0.042,Y -475.485,Z 295.358,A 0.000,B 0.000,C 90.000,E1 100.433} C_DIS
LIN {X -0.205,Y -476.129,Z 295.356,A 0.000,B 0.000,C 90.000,E1 100.141} C_DIS
LIN {X 0.078,Y -482.044,Z 295.330,A 0.000,B 0.000,C 90.000,E1 95.454} C_DIS
LIN {X -0.131,Y -485.477,Z 295.305,A 0.000,B 0.000,C 90.000,E1 90.859} C_DIS
LIN {X 0.076,Y -486.247,Z 295.283,A 0.000,B 0.000,C 90.000,E1 86.846} C_DIS
LIN {X -0.098,Y -486.386,Z 295.281,A 0.000,B 0.000,C 90.000,E1 86.560} C_DIS
LIN {X 0.212,Y -486.363,Z 295.279,A 0.000,B 0.000,C 90.000,E1 86.216} C_DIS
LIN {X -0.185,Y -484.690,Z 295.254,A 0.000,B 0.000,C 90.000,E1 81.659} C_DIS
LIN {X -0.170,Y -483.693,Z 295.248,A 0.000,B 0.000,C 90.000,E1 80.735} C_DIS
LIN {X 0.193,Y -480.625,Z 295.228,A 0.000,B 0.000,C 90.000,E1 76.992} C_DIS
LIN {X 0.051,Y -480.301,Z 295.226,A 0.000,B 0.000,C 90.000,E1 76.700} C_DIS
LIN {X 0.003,Y -474.203,Z 295.201,A 0.000,B 0.000,C 90.000,E1 72.127} C_DIS
LIN {X -0.043,Y -478.180,Z 295.192,A 0.000,B 0.000,C 90.000,E1 70.496} C_DIS
LIN {X -0.103,Y -483.770,Z 295.180,A 0.000,B 0.000,C 90.000,E1 68.337} C_DIS
LIN {X -0.048,Y -487.965,Z 295.171,A 0.000,B 0.000,C 90.000,E1 66.794} C_DIS
LIN {X -0.171,Y -492.165,Z 295.163,A 0.000,B 0.000,C 90.000,E1 65.281} C_DIS
LIN {X -0.218,Y -496.413,Z 295.154,A 0.000,B 0.000,C 90.000,E1 63.768} C_DIS
LIN {X -0.069,Y -502.489,Z 295.142,A 0.000,B 0.000,C 90.000,E1 61.641} C_DIS
LIN {X -0.284,Y -507.686,Z 295.132,A 0.000,B 0.000,C 90.000,E1 59.871} C_DIS
LIN {X -0.135,Y -512.954,Z 295.123,A 0.000,B 0.000,C 90.000,E1 58.074} C_DIS
LIN {X 0.041,Y -517.252,Z 295.114,A 0.000,B 0.000,C 90.000,E1 56.580} C_DIS
LIN {X 0.158,Y -521.380,Z 295.106,A 0.000,B 0.000,C 90.000,E1 55.102} C_DIS
LIN {X -0.334,Y -524.545,Z 295.100,A 0.000,B 0.000,C 90.000,E1 53.989} C_DIS
LIN {X 0.262,Y -527.531,Z 295.093,A 0.000,B 0.000,C 90.000,E1 52.763} C_DIS
LIN {X 0.145,Y -530.891,Z 295.085,A 0.000,B 0.000,C 90.000,E1 51.331} C_DIS
LIN {X 0.011,Y -533.353,Z 295.079,A 0.000,B 0.000,C 90.000,E1 50.194} C_DIS
LIN {X -0.081,Y -535.592,Z 295.073,A 0.000,B 0.000,C 90.000,E1 49.057} C_DIS
LIN {X -0.141,Y -537.526,Z 295.066,A 0.000,B 0.000,C 90.000,E1 47.919} C_DIS
LIN {X 0.217,Y -538.442,Z 295.063,A 0.000,B 0.000,C 90.000,E1 47.310} C_DIS
LIN {X 0.164,Y -540.284,Z 295.055,A 0.000,B 0.000,C 90.000,E1 45.891} C_DIS
LIN {X 0.141,Y -541.365,Z 295.049,A 0.000,B 0.000,C 90.000,E1 44.757} C_DIS
LIN {X 0.131,Y -542.142,Z 295.042,A 0.000,B 0.000,C 90.000,E1 43.623} C_DIS
LIN {X 0.140,Y -542.585,Z 295.038,A 0.000,B 0.000,C 90.000,E1 42.771} C_DIS
LIN {X -0.230,Y -543.044,Z 295.031,A 0.000,B 0.000,C 90.000,E1 41.676} C_DIS
LIN {X -0.190,Y -543.200,Z 295.025,A 0.000,B 0.000,C 90.000,E1 40.539} C_DIS
LIN {X 0.240,Y -543.141,Z 295.020,A 0.000,B 0.000,C 90.000,E1 39.644} C_DIS
LIN {X -0.065,Y -542.897,Z 295.014,A 0.000,B 0.000,C 90.000,E1 38.543} C_DIS
LIN {X 0.057,Y -542.356,Z 295.008,A 0.000,B 0.000,C 90.000,E1 37.397} C_DIS
LIN {X -0.263,Y -541.670,Z 295.002,A 0.000,B 0.000,C 90.000,E1 36.297} C_DIS
LIN {X 0.297,Y -540.527,Z 294.994,A 0.000,B 0.000,C 90.000,E1 34.818} C_DIS
LIN {X 0.066,Y -539.587,Z 294.987,A 0.000,B 0.000,C 90.000,E1 33.706} C_DIS
LIN {X -0.007,Y -537.691,Z 294.976,A 0.000,B 0.000,C 90.000,E1 31.720} C_DIS
LIN {X 0.066,Y -536.236,Z 294.968,A 0.000,B 0.000,C 90.000,E1 30.285} C_DIS
LIN {X -0.080,Y -534.762,Z 294.960,A 0.000,B 0.000,C 90.000,E1 28.871} C_DIS
LIN {X 0.131,Y -533.006,Z 294.951,A 0.000,B 0.000,C 90.000,E1 27.129} C_DIS
LIN {X -0.222,Y -530.961,Z 294.940,A 0.000,B 0.000,C 90.000,E1 25.155} C_DIS
LIN {X 0.030,Y -528.769,Z 294.927,A 0.000,B 0.000,C 90.000,E1 22.823} C_DIS
LIN {X 0.070,Y -527.795,Z 294.920,A 0.000,B 0.000,C 90.000,E1 21.663} C_DIS
LIN {X -0.199,Y -525.792,Z 294.906,A 0.000,B 0.000,C 90.000,E1 19.087} C_DIS
LIN {X -0.043,Y -524.406,Z 294.895,A 0.000,B 0.000,C 90.000,E1 17.040} C_DIS
LIN {X 0.071,Y -522.947,Z 294.879,A 0.000,B 0.000,C 90.000,E1 14.120} C_DIS
LIN {X 0.247,Y -522.088,Z 294.866,A 0.000,B 0.000,C 90.000,E1 11.771} C_DIS
LIN {X 0.286,Y -521.652,Z 294.854,A 0.000,B 0.000,C 90.000,E1 9.726} C_DIS
LIN {X 0.139,Y -521.514,Z 294.845,A 0.000,B 0.000,C 90.000,E1 7.992} C_DIS
LIN {X -0.139,Y -521.741,Z 294.828,A 0.000,B 0.000,C 90.000,E1 5.106} C_DIS
LIN {X 0.028,Y -522.550,Z 294.814,A 0.000,B 0.000,C 90.000,E1 2.465} C_DIS
LIN {X 0.000,Y -523.669,Z 294.800,A 0.000,B 0.000,C 90.000,E1 360.000} C_DIS
LIN {X -0.054,Y -525.303,Z 294.788,A 0.000,B 0.000,C 90.000,E1 357.764} C_DIS
LIN {X -0.244,Y -526.769,Z 294.778,A 0.000,B 0.000,C 90.000,E1 356.045} C_DIS
LIN {X 0.176,Y -529.151,Z 294.765,A 0.000,B 0.000,C 90.000,E1 353.685} C_DIS
LIN {X 0.026,Y -536.926,Z 294.738,A 0.000,B 0.000,C 90.000,E1 348.814} C_DIS
LIN {X -0.211,Y -543.649,Z 294.722,A 0.000,B 0.000,C 90.000,E1 345.992} C_DIS
LIN {X -0.088,Y -547.910,Z 294.713,A 0.000,B 0.000,C 90.000,E1 344.283} C_DIS
LIN {X 0.270,Y -553.973,Z 294.700,A 0.000,B 0.000,C 90.000,E1 342.000} C_DIS
LIN {X 0.056,Y -561.407,Z 294.686,A 0.000,B 0.000,C 90.000,E1 339.518} C_DIS
LIN {X 0.200,Y -566.772,Z 294.677,A 0.000,B 0.000,C 90.000,E1 337.847} C_DIS
LIN {X -0.061,Y -572.293,Z 294.668,A 0.000,B 0.000,C 90.000,E1 336.230} C_DIS
LIN {X 0.026,Y -577.919,Z 294.659,A 0.000,B 0.000,C 90.000,E1 334.588} C_DIS
LIN {X -0.295,Y -583.746,Z 294.650,A 0.000,B 0.000,C 90.000,E1 332.999} C_DIS
LIN {X -0.125,Y -588.411,Z 294.642,A 0.000,B 0.000,C 90.000,E1 331.641} C_DIS
LIN {X 0.122,Y -592.970,Z 294.635,A 0.000,B 0.000,C 90.000,E1 330.284} C_DIS
LIN {X -0.287,Y -597.441,Z 294.628,A 0.000,B 0.000,C 90.000,E1 328.997} C_DIS
LIN {X -0.103,Y -601.928,Z 294.620,A 0.000,B 0.000,C 90.000,E1 327.661} C_DIS
LIN {X -0.022,Y -606.566,Z 294.613,A 0.000,B 0.000,C 90.000,E1 326.342} C_DIS
LIN {X -0.130,Y -613.252,Z 294.603,A 0.000,B 0.000,C 90.000,E1 324.529} C_DIS
LIN {X -0.161,Y -616.945,Z 294.597,A 0.000,B 0.000,C 90.000,E1 323.497} C_DIS
LIN {X 0.045,Y -621.247,Z 294.590,A 0.000,B 0.000,C 90.000,E1 322.190} C_DIS
LIN {X -0.159,Y -625.219,Z 294.583,A 0.000,B 0.000,C 90.000,E1 320.928} C_DIS
LIN {X 0.186,Y -629.135,Z 294.576,A 0.000,B 0.000,C 90.000,E1 319.622} C_DIS
LIN {X 0.163,Y -632.150,Z 294.570,A 0.000,B 0.000,C 90.000,E1 318.609} C_DIS
LIN {X -0.345,Y -635.752,Z 294.563,A 0.000,B 0.000,C 90.000,E1 317.391} C_DIS
LIN {X 0.358,Y -640.850,Z 294.553,A 0.000,B 0.000,C 90.000,E1 315.567} C_DIS
LIN {X -0.113,Y -645.186,Z 294.545,A 0.000,B 0.000,C 90.000,E1 314.109} C_DIS
LIN {X 0.086,Y -647.931,Z 294.540,A 0.000,B 0.000,C 90.000,E1 313.095} C_DIS
LIN {X 0.268,Y -651.226,Z 294.533,A 0.000,B 0.000,C 90.000,E1 311.838} C_DIS
LIN {X 0.065,Y -654.186,Z 294.526,A 0.000,B 0.000,C 90.000,E1 310.620} C_DIS
LIN {X -0.050,Y -656.324,Z 294.520,A 0.000,B 0.000,C 90.000,E1 309.644} C_DIS
LIN {X -0.096,Y -657.798,Z 294.516,A 0.000,B 0.000,C 90.000,E1 308.910} C_DIS
LIN {X -0.172,Y -659.574,Z 294.511,A 0.000,B 0.000,C 90.000,E1 307.935} C_DIS
LIN {X -0.110,Y -661.113,Z 294.505,A 0.000,B 0.000,C 90.000,E1 306.950} C_DIS
LIN {X -0.019,Y -662.382,Z 294.500,A 0.000,B 0.000,C 90.000,E1 305.964} C_DIS
LIN {X -0.016,Y -663.032,Z 294.496,A 0.000,B 0.000,C 90.000,E1 305.231} C_DIS
LIN {X 0.150,Y -663.330,Z 294.492,A 0.000,B 0.000,C 90.000,E1 304.485} C_DIS
LIN {X 0.265,Y -663.600,Z 294.486,A 0.000,B 0.000,C 90.000,E1 303.499} C_DIS
LIN {X 0.010,Y -663.399,Z 294.481,A 0.000,B 0.000,C 90.000,E1 302.546} C_DIS
LIN {X 0.058,Y -663.184,Z 294.478,A 0.000,B 0.000,C 90.000,E1 302.054} C_DIS
LIN {X -0.118,Y -662.424,Z 294.474,A 0.000,B 0.000,C 90.000,E1 301.337} C_DIS
LIN {X 0.046,Y -661.383,Z 294.470,A 0.000,B 0.000,C 90.000,E1 300.590} C_DIS
LIN {X -0.136,Y -660.034,Z 294.466,A 0.000,B 0.000,C 90.000,E1 299.873} C_DIS
LIN {X 0.240,Y -657.370,Z 294.459,A 0.000,B 0.000,C 90.000,E1 298.615} C_DIS
LIN {X 0.252,Y -654.431,Z 294.452,A 0.000,B 0.000,C 90.000,E1 297.385} C_DIS
LIN {X -0.077,Y -651.300,Z 294.445,A 0.000,B 0.000,C 90.000,E1 296.181} C_DIS
LIN {X -0.082,Y -647.348,Z 294.437,A 0.000,B 0.000,C 90.000,E1 294.695} C_DIS
LIN {X -0.198,Y -643.963,Z 294.430,A 0.000,B 0.000,C 90.000,E1 293.462} C_DIS
LIN {X -0.109,Y -640.574,Z 294.423,A 0.000,B 0.000,C 90.000,E1 292.206} C_DIS
LIN {X 0.083,Y -636.663,Z 294.415,A 0.000,B 0.000,C 90.000,E1 290.684} C_DIS
LIN {X 0.034,Y -631.592,Z 294.404,A 0.000,B 0.000,C 90.000,E1 288.671} C_DIS
LIN {X -0.159,Y -627.398,Z 294.394,A 0.000,B 0.000,C 90.000,E1 286.913} C_DIS
LIN {X 0.129,Y -622.615,Z 294.381,A 0.000,B 0.000,C 90.000,E1 284.592} C_DIS
LIN {X 0.122,Y -617.726,Z 294.366,A 0.000,B 0.000,C 90.000,E1 281.771} C_DIS
LIN {X -0.053,Y -614.242,Z 294.351,A 0.000,B 0.000,C 90.000,E1 279.208} C_DIS
LIN {X -0.183,Y -611.077,Z 294.332,A 0.000,B 0.000,C 90.000,E1 275.853} C_DIS
LIN {X -0.015,Y -609.592,Z 294.317,A 0.000,B 0.000,C 90.000,E1 272.980} C_DIS
LIN {X 0.074,Y -609.109,Z 294.304,A 0.000,B 0.000,C 90.000,E1 270.630} C_DIS
LIN {X -0.131,Y -609.316,Z 294.292,A 0.000,B 0.000,C 90.000,E1 268.568} C_DIS
LIN {X 0.236,Y -611.104,Z 294.272,A 0.000,B 0.000,C 90.000,E1 264.894} C_DIS
LIN {X 0.242,Y -612.913,Z 294.260,A 0.000,B 0.000,C 90.000,E1 262.818} C_DIS
LIN {X -0.232,Y -615.207,Z 294.249,A 0.000,B 0.000,C 90.000,E1 260.792} C_DIS
LIN {X 0.056,Y -618.086,Z 294.237,A 0.000,B 0.000,C 90.000,E1 258.701} C_DIS
LIN {X -0.103,Y -620.396,Z 294.229,A 0.000,B 0.000,C 90.000,E1 257.173} C_DIS
LIN {X -0.214,Y -622.757,Z 294.220,A 0.000,B 0.000,C 90.000,E1 255.644} C_DIS
LIN {X 0.296,Y -624.253,Z 294.215,A 0.000,B 0.000,C 90.000,E1 254.574} C_DIS
LIN {X -0.165,Y -625.172,Z 294.210,A 0.000,B 0.000,C 90.000,E1 253.850} C_DIS
LIN {X -0.216,Y -626.088,Z 294.205,A 0.000,B 0.000,C 90.000,E1 252.834} C_DIS
LIN {X 0.124,Y -627.049,Z 294.198,A 0.000,B 0.000,C 90.000,E1 251.529} C_DIS
LIN {X -0.101,Y -627.483,Z 294.193,A 0.000,B 0.000,C 90.000,E1 250.786} C_DIS
LIN {X 0.067,Y -627.655,Z 294.188,A 0.000,B 0.000,C 90.000,E1 249.752} C_DIS
LIN {X -0.360,Y -627.576,Z 294.183,A 0.000,B 0.000,C 90.000,E1 249.028} C_DIS
LIN {X 0.017,Y -627.227,Z 294.179,A 0.000,B 0.000,C 90.000,E1 248.230} C_DIS
LIN {X -0.190,Y -626.657,Z 294.175,A 0.000,B 0.000,C 90.000,E1 247.486} C_DIS
LIN {X -0.156,Y -625.829,Z 294.171,A 0.000,B 0.000,C 90.000,E1 246.719} C_DIS
LIN {X 0.199,Y -624.759,Z 294.166,A 0.000,B 0.000,C 90.000,E1 245.921} C_DIS
LIN {X -0.031,Y -623.116,Z 294.161,A 0.000,B 0.000,C 90.000,E1 244.921} C_DIS
LIN {X -0.020,Y -621.576,Z 294.156,A 0.000,B 0.000,C 90.000,E1 244.152} C_DIS
LIN {X -0.032,Y -618.562,Z 294.149,A 0.000,B 0.000,C 90.000,E1 242.871} C_DIS
LIN {X -0.083,Y -615.857,Z 294.144,A 0.000,B 0.000,C 90.000,E1 241.847} C_DIS
LIN {X 0.118,Y -613.018,Z 294.138,A 0.000,B 0.000,C 90.000,E1 240.795} C_DIS
LIN {X -0.289,Y -609.306,Z 294.131,A 0.000,B 0.000,C 90.000,E1 239.537} C_DIS
LIN {X 0.076,Y -605.497,Z 294.123,A 0.000,B 0.000,C 90.000,E1 238.201} C_DIS
LIN {X 0.104,Y -600.793,Z 294.115,A 0.000,B 0.000,C 90.000,E1 236.628} C_DIS
LIN {X -0.334,Y -598.389,Z 294.110,A 0.000,B 0.000,C 90.000,E1 235.881} C_DIS
LIN {X 0.260,Y -595.019,Z 294.104,A 0.000,B 0.000,C 90.000,E1 234.769} C_DIS
LIN {X 0.318,Y -591.525,Z 294.099,A 0.000,B 0.000,C 90.000,E1 233.703} C_DIS
LIN {X -0.177,Y -584.680,Z 294.087,A 0.000,B 0.000,C 90.000,E1 231.618} C_DIS
LIN {X -0.180,Y -580.441,Z 294.079,A 0.000,B 0.000,C 90.000,E1 230.275} C_DIS
LIN {X -0.164,Y -572.793,Z 294.066,A 0.000,B 0.000,C 90.000,E1 227.838} C_DIS
LIN {X -0.001,Y -568.658,Z 294.058,A 0.000,B 0.000,C 90.000,E1 226.458} C_DIS
LIN {X -0.251,Y -563.528,Z 294.049,A 0.000,B 0.000,C 90.000,E1 224.838} C_DIS
LIN {X 0.054,Y -560.147,Z 294.043,A 0.000,B 0.000,C 90.000,E1 223.704} C_DIS
LIN {X -0.007,Y -555.996,Z 294.035,A 0.000,B 0.000,C 90.000,E1 222.324} C_DIS
LIN {X -0.076,Y -550.050,Z 294.024,A 0.000,B 0.000,C 90.000,E1 220.378} C_DIS
LIN {X 0.175,Y -544.016,Z 294.013,A 0.000,B 0.000,C 90.000,E1 218.382} C_DIS
LIN {X -0.127,Y -540.656,Z 294.007,A 0.000,B 0.000,C 90.000,E1 217.282} C_DIS
LIN {X -0.338,Y -534.682,Z 293.996,A 0.000,B 0.000,C 90.000,E1 215.311} C_DIS
LIN {X 0.088,Y -531.366,Z 293.990,A 0.000,B 0.000,C 90.000,E1 214.119} C_DIS
LIN {X -0.171,Y -523.435,Z 293.974,A 0.000,B 0.000,C 90.000,E1 211.258} C_DIS
LIN {X -0.051,Y -518.074,Z 293.962,A 0.000,B 0.000,C 90.000,E1 209.205} C_DIS
LIN {X 0.125,Y -514.487,Z 293.954,A 0.000,B 0.000,C 90.000,E1 207.719} C_DIS
LIN {X -0.047,Y -508.311,Z 293.939,A 0.000,B 0.000,C 90.000,E1 205.079} C_DIS
LIN {X 0.056,Y -502.589,Z 293.924,A 0.000,B 0.000,C 90.000,E1 202.386} C_DIS
LIN {X -0.075,Y -498.346,Z 293.913,A 0.000,B 0.000,C 90.000,E1 200.301} C_DIS
LIN {X -0.075,Y -493.414,Z 293.898,A 0.000,B 0.000,C 90.000,E1 197.583} C_DIS
LIN {X 0.080,Y -488.922,Z 293.882,A 0.000,B 0.000,C 90.000,E1 194.828} C_DIS
LIN {X -0.037,Y -486.167,Z 293.872,A 0.000,B 0.000,C 90.000,E1 193.008} C_DIS
LIN {X -0.207,Y -483.620,Z 293.862,A 0.000,B 0.000,C 90.000,E1 191.186} C_DIS
LIN {X -0.204,Y -480.819,Z 293.850,A 0.000,B 0.000,C 90.000,E1 189.029} C_DIS
LIN {X 0.048,Y -478.316,Z 293.838,A 0.000,B 0.000,C 90.000,E1 186.834} C_DIS
LIN {X 0.087,Y -476.652,Z 293.829,A 0.000,B 0.000,C 90.000,E1 185.277} C_DIS
LIN {X 0.128,Y -474.501,Z 293.817,A 0.000,B 0.000,C 90.000,E1 183.094} C_DIS
LIN {X 0.063,Y -472.600,Z 293.805,A 0.000,B 0.000,C 90.000,E1 180.917} C_DIS
LIN {X -0.051,Y -471.161,Z 293.793,A 0.000,B 0.000,C 90.000,E1 178.740} C_DIS
LIN {X -0.133,Y -469.780,Z 293.777,A 0.000,B 0.000,C 90.000,E1 175.927} C_DIS
LIN {X -0.221,Y -469.040,Z 293.762,A 0.000,B 0.000,C 90.000,E1 173.109} C_DIS
LIN {X -0.105,Y -468.840,Z 293.755,A 0.000,B 0.000,C 90.000,E1 171.837} C_DIS
LIN {X 0.186,Y -468.628,Z 293.741,A 0.000,B 0.000,C 90.000,E1 169.285} C_DIS
LIN {X -0.082,Y -469.044,Z 293.723,A 0.000,B 0.000,C 90.000,E1 166.172} C_DIS
LIN {X 0.037,Y -470.326,Z 293.706,A 0.000,B 0.000,C 90.000,E1 163.015} C_DIS
LIN {X 0.038,Y -472.398,Z 293.688,A 0.000,B 0.000,C 90.000,E1 159.880} C_DIS
LIN {X 0.242,Y -474.169,Z 293.676,A 0.000,B 0.000,C 90.000,E1 157.667} C_DIS
LIN {X -0.247,Y -477.053,Z 293.661,A 0.000,B 0.000,C 90.000,E1 154.921} C_DIS
LIN {X -0.271,Y -481.483,Z 293.642,A 0.000,B 0.000,C 90.000,E1 151.513} C_DIS
LIN {X 0.124,Y -484.458,Z 293.631,A 0.000,B 0.000,C 90.000,E1 149.616} C_DIS
LIN {X 0.237,Y -488.145,Z 293.619,A 0.000,B 0.000,C 90.000,E1 147.454} C_DIS
LIN {X -0.213,Y -491.439,Z 293.609,A 0.000,B 0.000,C 90.000,E1 145.674} C_DIS
LIN {X -0.029,Y -494.695,Z 293.599,A 0.000,B 0.000,C 90.000,E1 143.829} C_DIS
LIN {X -0.195,Y -496.821,Z 293.592,A 0.000,B 0.000,C 90.000,E1 142.637} C_DIS
LIN {X 0.146,Y -499.371,Z 293.584,A 0.000,B 0.000,C 90.000,E1 141.090} C_DIS
LIN {X 0.082,Y -500.757,Z 293.579,A 0.000,B 0.000,C 90.000,E1 140.194} C_DIS
LIN {X -0.091,Y -502.432,Z 293.572,A 0.000,B 0.000,C 90.000,E1 139.013} C_DIS
LIN {X 0.207,Y -503.585,Z 293.567,A 0.000,B 0.000,C 90.000,E1 138.081} C_DIS
LIN {X -0.192,Y -504.448,Z 293.562,A 0.000,B 0.000,C 90.000,E1 137.229} C_DIS
LIN {X 0.129,Y -505.098,Z 293.557,A 0.000,B 0.000,C 90.000,E1 136.296} C_DIS
LIN {X -0.036,Y -505.518,Z 293.551,A 0.000,B 0.000,C 90.000,E1 135.121} C_DIS
LIN {X 0.292,Y -505.590,Z 293.546,A 0.000,B 0.000,C 90.000,E1 134.190} C_DIS
LIN {X -0.088,Y -505.407,Z 293.541,A 0.000,B 0.000,C 90.000,E1 133.338} C_DIS
LIN {X -0.124,Y -504.910,Z 293.536,A 0.000,B 0.000,C 90.000,E1 132.447} C_DIS
LIN {X 0.202,Y -504.209,Z 293.531,A 0.000,B 0.000,C 90.000,E1 131.515} C_DIS
LIN {X 0.186,Y -503.309,Z 293.526,A 0.000,B 0.000,C 90.000,E1 130.620} C_DIS
LIN {X 0.049,Y -501.814,Z 293.519,A 0.000,B 0.000,C 90.000,E1 129.439} C_DIS
LIN {X -0.046,Y -499.376,Z 293.509,A 0.000,B 0.000,C 90.000,E1 127.649} C_DIS
LIN {X 0.013,Y -497.064,Z 293.501,A 0.000,B 0.000,C 90.000,E1 126.137} C_DIS
LIN {X -0.125,Y -495.022,Z 293.494,A 0.000,B 0.000,C 90.000,E1 124.945} C_DIS
LIN {X 0.221,Y -491.625,Z 293.484,A 0.000,B 0.000,C 90.000,E1 123.086} C_DIS
LIN {X 0.144,Y -489.318,Z 293.477,A 0.000,B 0.000,C 90.000,E1 121.878} C_DIS
LIN {X -0.145,Y -486.375,Z 293.469,A 0.000,B 0.000,C 90.000,E1 120.384} C_DIS
LIN {X 0.105,Y -483.378,Z 293.460,A 0.000,B 0.000,C 90.000,E1 118.821} C_DIS
LIN {X -0.127,Y -480.363,Z 293.452,A 0.000,B 0.000,C 90.000,E1 117.308} C_DIS
LIN {X 0.214,Y -477.357,Z 293.443,A 0.000,B 0.000,C 90.000,E1 115.720} C_DIS
LIN {X -0.133,Y -474.349,Z 293.434,A 0.000,B 0.000,C 90.000,E1 114.207} C_DIS
LIN {X -0.178,Y -470.182,Z 293.422,A 0.000,B 0.000,C 90.000,E1 112.025} C_DIS
LIN {X -0.080,Y -466.141,Z 293.410,A 0.000,B 0.000,C 90.000,E1 109.812} C_DIS
LIN {X 0.037,Y -462.392,Z 293.398,A 0.000,B 0.000,C 90.000,E1 107.583} C_DIS
LIN {X 0.141,Y -462.030,Z 293.397,A 0.000,B 0.000,C 90.000,E1 107.347} C_DIS
LIN {X 0.101,Y -462.025,Z 293.396,A 0.000,B 0.000,C 90.000,E1 107.347} C_DIS
LIN {X -0.101,Y -467.393,Z 293.384,A 0.000,B 0.000,C 90.000,E1 105.064} C_DIS
LIN {X 0.155,Y -468.031,Z 293.382,A 0.000,B 0.000,C 90.000,E1 104.717} C_DIS
LIN {X 0.133,Y -476.240,Z 293.356,A 0.000,B 0.000,C 90.000,E1 100.018} C_DIS
LIN {X -0.082,Y -482.134,Z 293.330,A 0.000,B 0.000,C 90.000,E1 95.391} C_DIS
LIN {X 0.153,Y -485.530,Z 293.304,A 0.000,B 0.000,C 90.000,E1 90.745} C_DIS
LIN {X 0.185,Y -486.379,Z 293.280,A 0.000,B 0.000,C 90.000,E1 86.445} C_DIS
LIN {X 0.009,Y -486.349,Z 293.279,A 0.000,B 0.000,C 90.000,E1 86.159} C_DIS
LIN {X 0.088,Y -484.662,Z 293.253,A 0.000,B 0.000,C 90.000,E1 81.546} C_DIS
LIN {X -0.022,Y -480.581,Z 293.227,A 0.000,B 0.000,C 90.000,E1 76.937} C_DIS
LIN {X 0.157,Y -479.652,Z 293.224,A 0.000,B 0.000,C 90.000,E1 76.297} C_DIS
LIN {X 0.177,Y -473.990,Z 293.200,A 0.000,B 0.000,C 90.000,E1 71.945} C_DIS
LIN {X -0.146,Y -473.910,Z 293.200,A 0.000,B 0.000,C 90.000,E1 71.945} C_DIS
LIN {X -0.186,Y -473.902,Z 293.200,A 0.000,B 0.000,C 90.000,E1 71.945} C_DIS
LIN {X -0.126,Y -477.637,Z 293.191,A 0.000,B 0.000,C 90.000,E1 70.423} C_DIS
LIN {X 0.080,Y -484.049,Z 293.177,A 0.000,B 0.000,C 90.000,E1 67.922} C_DIS
LIN {X -0.123,Y -488.208,Z 293.169,A 0.000,B 0.000,C 90.000,E1 66.410} C_DIS
LIN {X -0.028,Y -491.587,Z 293.162,A 0.000,B 0.000,C 90.000,E1 65.177} C_DIS
LIN {X 0.124,Y -495.852,Z 293.154,A 0.000,B 0.000,C 90.000,E1 63.640} C_DIS
LIN {X 0.262,Y -501.921,Z 293.142,A 0.000,B 0.000,C 90.000,E1 61.513} C_DIS
LIN {X 0.035,Y -507.123,Z 293.132,A 0.000,B 0.000,C 90.000,E1 59.744} C_DIS
LIN {X -0.262,Y -512.378,Z 293.122,A 0.000,B 0.000,C 90.000,E1 57.995} C_DIS
LIN {X -0.094,Y -516.675,Z 293.114,A 0.000,B 0.000,C 90.000,E1 56.501} C_DIS
LIN {X 0.015,Y -520.809,Z 293.106,A 0.000,B 0.000,C 90.000,E1 55.022} C_DIS
LIN {X -0.060,Y -523.966,Z 293.099,A 0.000,B 0.000,C 90.000,E1 53.863} C_DIS
LIN {X 0.105,Y -526.940,Z 293.093,A 0.000,B 0.000,C 90.000,E1 52.683} C_DIS
LIN {X -0.022,Y -530.295,Z 293.085,A 0.000,B 0.000,C 90.000,E1 51.251} C_DIS
LIN {X 0.245,Y -532.709,Z 293.078,A 0.000,B 0.000,C 90.000,E1 50.070} C_DIS
LIN {X 0.139,Y -534.944,Z 293.072,A 0.000,B 0.000,C 90.000,E1 48.933} C_DIS
LIN {X 0.064,Y -536.823,Z 293.066,A 0.000,B 0.000,C 90.000,E1 47.796} C_DIS
LIN {X 0.014,Y -538.100,Z 293.061,A 0.000,B 0.000,C 90.000,E1 46.944} C_DIS
LIN {X -0.047,Y -539.545,Z 293.055,A 0.000,B 0.000,C 90.000,E1 45.810} C_DIS
LIN {X -0.081,Y -540.571,Z 293.048,A 0.000,B 0.000,C 90.000,E1 44.676} C_DIS
LIN {X -0.104,Y -541.319,Z 293.042,A 0.000,B 0.000,C 90.000,E1 43.542} C_DIS
LIN {X -0.104,Y -541.749,Z 293.037,A 0.000,B 0.000,C 90.000,E1 42.690} C_DIS
LIN {X -0.081,Y -542.163,Z 293.031,A 0.000,B 0.000,C 90.000,E1 41.553} C_DIS
LIN {X -0.070,Y -542.288,Z 293.026,A 0.000,B 0.000,C 90.000,E1 40.701} C_DIS
LIN {X -0.065,Y -542.279,Z 293.021,A 0.000,B 0.000,C 90.000,E1 39.850} C_DIS
LIN {X 0.037,Y -542.015,Z 293.015,A 0.000,B 0.000,C 90.000,E1 38.705} C_DIS
LIN {X 0.025,Y -541.667,Z 293.010,A 0.000,B 0.000,C 90.000,E1 37.855} C_DIS
LIN {X 0.122,Y -541.024,Z 293.004,A 0.000,B 0.000,C 90.000,E1 36.710} C_DIS
LIN {X -0.130,Y -540.440,Z 292.999,A 0.000,B 0.000,C 90.000,E1 35.884} C_DIS
LIN {X -0.326,Y -539.005,Z 292.990,A 0.000,B 0.000,C 90.000,E1 34.199} C_DIS
LIN {X -0.128,Y -537.924,Z 292.984,A 0.000,B 0.000,C 90.000,E1 33.038} C_DIS
LIN {X 0.053,Y -536.598,Z 292.976,A 0.000,B 0.000,C 90.000,E1 31.592} C_DIS
LIN {X 0.093,Y -534.814,Z 292.966,A 0.000,B 0.000,C 90.000,E1 29.873} C_DIS
LIN {X 0.092,Y -533.016,Z 292.957,A 0.000,B 0.000,C 90.000,E1 28.153} C_DIS
LIN {X -0.054,Y -532.175,Z 292.952,A 0.000,B 0.000,C 90.000,E1 27.308} C_DIS
LIN {X -0.252,Y -529.766,Z 292.939,A 0.000,B 0.000,C 90.000,E1 25.027} C_DIS
LIN {X -0.036,Y -527.580,Z 292.926,A 0.000,B 0.000,C 90.000,E1 22.695} C_DIS
LIN {X -0.017,Y -526.585,Z 292.920,A 0.000,B 0.000,C 90.000,E1 21.535} C_DIS
LIN {X 0.167,Y -524.587,Z 292.905,A 0.000,B 0.000,C 90.000,E1 18.906} C_DIS
LIN {X 0.137,Y -523.362,Z 292.896,A 0.000,B 0.000,C 90.000,E1 17.166} C_DIS
LIN {X 0.221,Y -521.948,Z 292.881,A 0.000,B 0.000,C 90.000,E1 14.537} C_DIS
LIN {X -0.146,Y -521.336,Z 292.873,A 0.000,B 0.000,C 90.000,E1 13.119} C_DIS
LIN {X -0.119,Y -520.565,Z 292.858,A 0.000,B 0.000,C 90.000,E1 10.489} C_DIS
LIN {X -0.208,Y -520.286,Z 292.845,A 0.000,B 0.000,C 90.000,E1 8.163} C_DIS
LIN {X -0.084,Y -520.486,Z 292.827,A 0.000,B 0.000,C 90.000,E1 4.935} C_DIS
LIN {X 0.045,Y -521.314,Z 292.813,A 0.000,B 0.000,C 90.000,E1 2.293} C_DIS
LIN {X -0.022,Y -523.507,Z 292.791,A 0.000,B 0.000,C 90.000,E1 358.339} C_DIS
LIN {X 0.215,Y -525.422,Z 292.778,A 0.000,B 0.000,C 90.000,E1 355.988} C_DIS
LIN {X 0.088,Y -528.114,Z 292.763,A 0.000,B 0.000,C 90.000,E1 353.394} C_DIS
LIN {X -0.111,Y -536.159,Z 292.736,A 0.000,B 0.000,C 90.000,E1 348.522} C_DIS
LIN {X 0.073,Y -542.290,Z 292.722,A 0.000,B 0.000,C 90.000,E1 345.936} C_DIS
LIN {X 0.313,Y -546.557,Z 292.713,A 0.000,B 0.000,C 90.000,E1 344.212} C_DIS
LIN {X -0.312,Y -551.858,Z 292.702,A 0.000,B 0.000,C 90.000,E1 342.308} C_DIS
LIN {X -0.219,Y -561.870,Z 292.683,A 0.000,B 0.000,C 90.000,E1 338.954} C_DIS
LIN {X 0.055,Y -568.223,Z 292.672,A 0.000,B 0.000,C 90.000,E1 336.997} C_DIS
LIN {X 0.045,Y -573.857,Z 292.663,A 0.000,B 0.000,C 90.000,E1 335.357} C_DIS
LIN {X -0.128,Y -581.544,Z 292.651,A 0.000,B 0.000,C 90.000,E1 333.204} C_DIS
LIN {X -0.001,Y -586.268,Z 292.644,A 0.000,B 0.000,C 90.000,E1 331.847} C_DIS
LIN {X -0.126,Y -591.727,Z 292.635,A 0.000,B 0.000,C 90.000,E1 330.255} C_DIS
LIN {X -0.132,Y -597.099,Z 292.626,A 0.000,B 0.000,C 90.000,E1 328.663} C_DIS
LIN {X -0.304,Y -603.500,Z 292.616,A 0.000,B 0.000,C 90.000,E1 326.834} C_DIS
LIN {X 0.005,Y -610.151,Z 292.605,A 0.000,B 0.000,C 90.000,E1 324.975} C_DIS
LIN {X -0.272,Y -614.857,Z 292.598,A 0.000,B 0.000,C 90.000,E1 323.703} C_DIS
LIN {X 0.078,Y -618.420,Z 292.593,A 0.000,B 0.000,C 90.000,E1 322.637} C_DIS
LIN {X -0.336,Y -620.943,Z 292.588,A 0.000,B 0.000,C 90.000,E1 321.904} C_DIS
LIN {X -0.064,Y -624.965,Z 292.581,A 0.000,B 0.000,C 90.000,E1 320.598} C_DIS
LIN {X 0.194,Y -628.885,Z 292.574,A 0.000,B 0.000,C 90.000,E1 319.299} C_DIS
LIN {X 0.105,Y -632.579,Z 292.567,A 0.000,B 0.000,C 90.000,E1 318.038} C_DIS
LIN {X -0.078,Y -636.891,Z 292.559,A 0.000,B 0.000,C 90.000,E1 316.539} C_DIS
LIN {X 0.362,Y -640.535,Z 292.552,A 0.000,B 0.000,C 90.000,E1 315.243} C_DIS
LIN {X -0.041,Y -644.146,Z 292.545,A 0.000,B 0.000,C 90.000,E1 314.028} C_DIS
LIN {X 0.076,Y -647.565,Z 292.538,A 0.000,B 0.000,C 90.000,E1 312.771} C_DIS
LIN {X 0.307,Y -650.181,Z 292.532,A 0.000,B 0.000,C 90.000,E1 311.757} C_DIS
LIN {X 0.031,Y -653.667,Z 292.524,A 0.000,B 0.000,C 90.000,E1 310.297} C_DIS
LIN {X -0.096,Y -655.740,Z 292.518,A 0.000,B 0.000,C 90.000,E1 309.322} C_DIS
LIN {X -0.096,Y -657.589,Z 292.513,A 0.000,B 0.000,C 90.000,E1 308.338} C_DIS
LIN {X -0.176,Y -659.186,Z 292.508,A 0.000,B 0.000,C 90.000,E1 307.363} C_DIS
LIN {X -0.116,Y -660.578,Z 292.502,A 0.000,B 0.000,C 90.000,E1 306.377} C_DIS
LIN {X -0.077,Y -661.143,Z 292.499,A 0.000,B 0.000,C 90.000,E1 305.884} C_DIS
LIN {X -0.032,Y -661.611,Z 292.497,A 0.000,B 0.000,C 90.000,E1 305.391} C_DIS
LIN {X 0.062,Y -661.996,Z 292.491,A 0.000,B 0.000,C 90.000,E1 304.405} C_DIS
LIN {X 0.156,Y -662.257,Z 292.486,A 0.000,B 0.000,C 90.000,E1 303.420} C_DIS
LIN {X -0.119,Y -661.983,Z 292.480,A 0.000,B 0.000,C 90.000,E1 302.467} C_DIS
LIN {X 0.128,Y -661.696,Z 292.478,A 0.000,B 0.000,C 90.000,E1 301.957} C_DIS
LIN {X -0.274,Y -660.908,Z 292.474,A 0.000,B 0.000,C 90.000,E1 301.258} C_DIS
LIN {X -0.128,Y -659.835,Z 292.470,A 0.000,B 0.000,C 90.000,E1 300.512} C_DIS
LIN {X 0.244,Y -658.451,Z 292.465,A 0.000,B 0.000,C 90.000,E1 299.745} C_DIS
LIN {X -0.297,Y -655.719,Z 292.459,A 0.000,B 0.000,C 90.000,E1 298.565} C_DIS
LIN {X -0.004,Y -652.746,Z 292.452,A 0.000,B 0.000,C 90.000,E1 297.308} C_DIS
LIN {X 0.121,Y -650.278,Z 292.446,A 0.000,B 0.000,C 90.000,E1 296.309} C_DIS
LIN {X -0.090,Y -645.644,Z 292.437,A 0.000,B 0.000,C 90.000,E1 294.591} C_DIS
LIN {X 0.033,Y -642.233,Z 292.430,A 0.000,B 0.000,C 90.000,E1 293.334} C_DIS
LIN {X -0.051,Y -637.545,Z 292.420,A 0.000,B 0.000,C 90.000,E1 291.589} C_DIS
LIN {X 0.275,Y -634.324,Z 292.413,A 0.000,B 0.000,C 90.000,E1 290.301} C_DIS
LIN {X -0.054,Y -629.308,Z 292.402,A 0.000,B 0.000,C 90.000,E1 288.308} C_DIS
LIN {X 0.017,Y -622.535,Z 292.385,A 0.000,B 0.000,C 90.000,E1 285.245} C_DIS
LIN {X 0.144,Y -617.350,Z 292.369,A 0.000,B 0.000,C 90.000,E1 282.411} C_DIS
LIN {X -0.298,Y -613.388,Z 292.353,A 0.000,B 0.000,C 90.000,E1 279.613} C_DIS
LIN {X -0.135,Y -609.843,Z 292.333,A 0.000,B 0.000,C 90.000,E1 275.967} C_DIS
LIN {X -0.018,Y -608.314,Z 292.317,A 0.000,B 0.000,C 90.000,E1 273.094} C_DIS
LIN {X 0.243,Y -607.834,Z 292.300,A 0.000,B 0.000,C 90.000,E1 269.943} C_DIS
LIN {X 0.136,Y -609.035,Z 292.278,A 0.000,B 0.000,C 90.000,E1 266.045} C_DIS
LIN {X -0.265,Y -610.812,Z 292.265,A 0.000,B 0.000,C 90.000,E1 263.742} C_DIS
LIN {X 0.070,Y -613.224,Z 292.252,A 0.000,B 0.000,C 90.000,E1 261.376} C_DIS
LIN {X -0.179,Y -616.721,Z 292.238,A 0.000,B 0.000,C 90.000,E1 258.814} C_DIS
LIN {X 0.243,Y -619.046,Z 292.229,A 0.000,B 0.000,C 90.000,E1 257.229} C_DIS
LIN {X 0.111,Y -621.414,Z 292.221,A 0.000,B 0.000,C 90.000,E1 255.700} C_DIS
LIN {X 0.003,Y -622.948,Z 292.215,A 0.000,B 0.000,C 90.000,E1 254.685} C_DIS
LIN {X -0.039,Y -623.892,Z 292.211,A 0.000,B 0.000,C 90.000,E1 253.921} C_DIS
LIN {X -0.115,Y -624.846,Z 292.205,A 0.000,B 0.000,C 90.000,E1 252.906} C_DIS
LIN {X 0.179,Y -625.975,Z 292.197,A 0.000,B 0.000,C 90.000,E1 251.348} C_DIS
LIN {X -0.056,Y -626.364,Z 292.192,A 0.000,B 0.000,C 90.000,E1 250.604} C_DIS
LIN {X -0.124,Y -626.461,Z 292.185,A 0.000,B 0.000,C 90.000,E1 249.337} C_DIS
LIN {X 0.241,Y -626.191,Z 292.181,A 0.000,B 0.000,C 90.000,E1 248.539} C_DIS
LIN {X 0.030,Y -625.533,Z 292.175,A 0.000,B 0.000,C 90.000,E1 247.539} C_DIS
LIN {X -0.191,Y -624.725,Z 292.171,A 0.000,B 0.000,C 90.000,E1 246.794} C_DIS
LIN {X 0.148,Y -623.675,Z 292.167,A 0.000,B 0.000,C 90.000,E1 245.997} C_DIS
LIN {X 0.162,Y -622.043,Z 292.161,A 0.000,B 0.000,C 90.000,E1 244.973} C_DIS
LIN {X 0.165,Y -620.524,Z 292.157,A 0.000,B 0.000,C 90.000,E1 244.204} C_DIS
LIN {X -0.129,Y -618.138,Z 292.151,A 0.000,B 0.000,C 90.000,E1 243.204} C_DIS
LIN {X 0.116,Y -616.216,Z 292.147,A 0.000,B 0.000,C 90.000,E1 242.410} C_DIS
LIN {X 0.006,Y -612.784,Z 292.140,A 0.000,B 0.000,C 90.000,E1 241.129} C_DIS
LIN {X 0.120,Y -609.121,Z 292.132,A 0.000,B 0.000,C 90.000,E1 239.822} C_DIS
LIN {X -0.108,Y -604.558,Z 292.124,A 0.000,B 0.000,C 90.000,E1 238.280} C_DIS
LIN {X -0.103,Y -599.850,Z 292.115,A 0.000,B 0.000,C 90.000,E1 236.707} C_DIS
LIN {X -0.317,Y -596.609,Z 292.109,A 0.000,B 0.000,C 90.000,E1 235.674} C_DIS
LIN {X -0.234,Y -593.214,Z 292.103,A 0.000,B 0.000,C 90.000,E1 234.609} C_DIS
LIN {X 0.016,Y -588.789,Z 292.096,A 0.000,B 0.000,C 90.000,E1 233.256} C_DIS
LIN {X -0.088,Y -583.750,Z 292.087,A 0.000,B 0.000,C 90.000,E1 231.662} C_DIS
LIN {X -0.023,Y -579.510,Z 292.080,A 0.000,B 0.000,C 90.000,E1 230.312} C_DIS
LIN {X -0.056,Y -571.883,Z 292.066,A 0.000,B 0.000,C 90.000,E1 227.877} C_DIS
LIN {X 0.059,Y -567.728,Z 292.058,A 0.000,B 0.000,C 90.000,E1 226.500} C_DIS
LIN {X 0.198,Y -562.574,Z 292.049,A 0.000,B 0.000,C 90.000,E1 224.838} C_DIS
LIN {X -0.305,Y -559.201,Z 292.043,A 0.000,B 0.000,C 90.000,E1 223.785} C_DIS
LIN {X 0.060,Y -554.144,Z 292.034,A 0.000,B 0.000,C 90.000,E1 222.081} C_DIS
LIN {X -0.049,Y -549.036,Z 292.025,A 0.000,B 0.000,C 90.000,E1 220.415} C_DIS
LIN {X -0.236,Y -543.003,Z 292.014,A 0.000,B 0.000,C 90.000,E1 218.463} C_DIS
LIN {X -0.118,Y -539.627,Z 292.007,A 0.000,B 0.000,C 90.000,E1 217.317} C_DIS
LIN {X -0.031,Y -533.662,Z 291.996,A 0.000,B 0.000,C 90.000,E1 215.311} C_DIS
LIN {X 0.065,Y -529.473,Z 291.988,A 0.000,B 0.000,C 90.000,E1 213.865} C_DIS
LIN {X 0.077,Y -522.356,Z 291.974,A 0.000,B 0.000,C 90.000,E1 211.258} C_DIS
LIN {X 0.128,Y -518.501,Z 291.966,A 0.000,B 0.000,C 90.000,E1 209.795} C_DIS
LIN {X 0.210,Y -514.129,Z 291.956,A 0.000,B 0.000,C 90.000,E1 208.025} C_DIS
LIN {X 0.111,Y -507.224,Z 291.939,A 0.000,B 0.000,C 90.000,E1 205.079} C_DIS
LIN {X -0.096,Y -502.121,Z 291.926,A 0.000,B 0.000,C 90.000,E1 202.717} C_DIS
LIN {X -0.044,Y -497.879,Z 291.915,A 0.000,B 0.000,C 90.000,E1 200.610} C_DIS
LIN {X 0.075,Y -495.026,Z 291.906,A 0.000,B 0.000,C 90.000,E1 199.087} C_DIS
LIN {X -0.096,Y -491.373,Z 291.894,A 0.000,B 0.000,C 90.000,E1 196.985} C_DIS
LIN {X -0.017,Y -487.471,Z 291.881,A 0.000,B 0.000,C 90.000,E1 194.537} C_DIS
LIN {X -0.035,Y -485.184,Z 291.872,A 0.000,B 0.000,C 90.000,E1 193.008} C_DIS
LIN {X -0.228,Y -482.667,Z 291.862,A 0.000,B 0.000,C 90.000,E1 191.186} C_DIS
LIN {X 0.225,Y -479.929,Z 291.850,A 0.000,B 0.000,C 90.000,E1 188.973} C_DIS
LIN {X -0.020,Y -477.455,Z 291.838,A 0.000,B 0.000,C 90.000,E1 186.834} C_DIS
LIN {X 0.003,Y -475.820,Z 291.829,A 0.000,B 0.000,C 90.000,E1 185.277} C_DIS
LIN {X -0.194,Y -473.430,Z 291.816,A 0.000,B 0.000,C 90.000,E1 182.808} C_DIS
LIN {X -0.028,Y -471.402,Z 291.802,A 0.000,B 0.000,C 90.000,E1 180.286} C_DIS
LIN {X -0.161,Y -470.121,Z 291.789,A 0.000,B 0.000,C 90.000,E1 178.108} C_DIS
LIN {X -0.035,Y -468.791,Z 291.772,A 0.000,B 0.000,C 90.000,E1 174.951} C_DIS
LIN {X -0.138,Y -468.345,Z 291.760,A 0.000,B 0.000,C 90.000,E1 172.761} C_DIS
LIN {X -0.031,Y -468.123,Z 291.753,A 0.000,B 0.000,C 90.000,E1 171.489} C_DIS
LIN {X -0.222,Y -467.994,Z 291.739,A 0.000,B 0.000,C 90.000,E1 168.993} C_DIS
LIN {X 0.127,Y -468.379,Z 291.723,A 0.000,B 0.000,C 90.000,E1 166.117} C_DIS
LIN {X 0.214,Y -469.674,Z 291.706,A 0.000,B 0.000,C 90.000,E1 162.960} C_DIS
LIN {X 0.181,Y -471.727,Z 291.688,A 0.000,B 0.000,C 90.000,E1 159.826} C_DIS
LIN {X -0.110,Y -473.784,Z 291.674,A 0.000,B 0.000,C 90.000,E1 157.358} C_DIS
LIN {X 0.018,Y -476.772,Z 291.659,A 0.000,B 0.000,C 90.000,E1 154.537} C_DIS
LIN {X -0.196,Y -480.352,Z 291.643,A 0.000,B 0.000,C 90.000,E1 151.769} C_DIS
LIN {X 0.177,Y -483.288,Z 291.633,A 0.000,B 0.000,C 90.000,E1 149.871} C_DIS
LIN {X -0.174,Y -487.415,Z 291.619,A 0.000,B 0.000,C 90.000,E1 147.454} C_DIS
LIN {X 0.039,Y -490.676,Z 291.609,A 0.000,B 0.000,C 90.000,E1 145.595} C_DIS
LIN {X -0.082,Y -493.896,Z 291.599,A 0.000,B 0.000,C 90.000,E1 143.783} C_DIS
LIN {X -0.104,Y -496.521,Z 291.590,A 0.000,B 0.000,C 90.000,E1 142.271} C_DIS
LIN {X 0.050,Y -498.541,Z 291.584,A 0.000,B 0.000,C 90.000,E1 141.045} C_DIS
LIN {X -0.028,Y -499.913,Z 291.579,A 0.000,B 0.000,C 90.000,E1 140.150} C_DIS
LIN {X 0.109,Y -501.602,Z 291.572,A 0.000,B 0.000,C 90.000,E1 138.933} C_DIS
LIN {X 0.061,Y -502.719,Z 291.567,A 0.000,B 0.000,C 90.000,E1 138.038} C_DIS
LIN {X -0.009,Y -503.597,Z 291.562,A 0.000,B 0.000,C 90.000,E1 137.148} C_DIS
LIN {X 0.303,Y -504.221,Z 291.557,A 0.000,B 0.000,C 90.000,E1 136.215} C_DIS
LIN {X -0.232,Y -504.651,Z 291.550,A 0.000,B 0.000,C 90.000,E1 135.081} C_DIS
LIN {X -0.270,Y -504.703,Z 291.545,A 0.000,B 0.000,C 90.000,E1 134.190} C_DIS
LIN {X 0.054,Y -504.512,Z 291.540,A 0.000,B 0.000,C 90.000,E1 133.257} C_DIS
LIN {X 0.008,Y -504.018,Z 291.535,A 0.000,B 0.000,C 90.000,E1 132.366} C_DIS
LIN {X -0.011,Y -503.309,Z 291.530,A 0.000,B 0.000,C 90.000,E1 131.472} C_DIS
LIN {X 0.296,Y -502.413,Z 291.525,A 0.000,B 0.000,C 90.000,E1 130.539} C_DIS
LIN {X 0.144,Y -500.945,Z 291.519,A 0.000,B 0.000,C 90.000,E1 129.358} C_DIS
LIN {X 0.026,Y -498.461,Z 291.509,A 0.000,B 0.000,C 90.000,E1 127.569} C_DIS
LIN {X -0.226,Y -496.150,Z 291.500,A 0.000,B 0.000,C 90.000,E1 126.091} C_DIS
LIN {X -0.089,Y -494.086,Z 291.494,A 0.000,B 0.000,C 90.000,E1 124.865} C_DIS
LIN {X -0.037,Y -490.678,Z 291.484,A 0.000,B 0.000,C 90.000,E1 123.038} C_DIS
LIN {X -0.036,Y -487.774,Z 291.475,A 0.000,B 0.000,C 90.000,E1 121.514} C_DIS
LIN {X 0.246,Y -485.447,Z 291.468,A 0.000,B 0.000,C 90.000,E1 120.256} C_DIS
LIN {X 0.040,Y -481.833,Z 291.458,A 0.000,B 0.000,C 90.000,E1 118.437} C_DIS
LIN {X 0.005,Y -479.443,Z 291.451,A 0.000,B 0.000,C 90.000,E1 117.206} C_DIS
LIN {X -0.091,Y -476.440,Z 291.443,A 0.000,B 0.000,C 90.000,E1 115.668} C_DIS
LIN {X 0.179,Y -473.443,Z 291.434,A 0.000,B 0.000,C 90.000,E1 114.079} C_DIS
LIN {X 0.105,Y -469.287,Z 291.422,A 0.000,B 0.000,C 90.000,E1 111.897} C_DIS
LIN {X 0.233,Y -465.862,Z 291.411,A 0.000,B 0.000,C 90.000,E1 109.993} C_DIS
LIN {X 0.221,Y -461.649,Z 291.397,A 0.000,B 0.000,C 90.000,E1 107.511} C_DIS
LIN {X 0.181,Y -461.656,Z 291.397,A 0.000,B 0.000,C 90.000,E1 107.511} C_DIS
LIN {X -0.005,Y -467.643,Z 291.383,A 0.000,B 0.000,C 90.000,E1 104.954} C_DIS
LIN {X -0.082,Y -469.567,Z 291.376,A 0.000,B 0.000,C 90.000,E1 103.703} C_DIS
LIN {X -0.048,Y -475.862,Z 291.357,A 0.000,B 0.000,C 90.000,E1 100.254} C_DIS
LIN {X -0.209,Y -476.332,Z 291.355,A 0.000,B 0.000,C 90.000,E1 99.962} C_DIS
LIN {X 0.217,Y -481.835,Z 291.331,A 0.000,B 0.000,C 90.000,E1 95.568} C_DIS
LIN {X 0.064,Y -482.183,Z 291.329,A 0.000,B 0.000,C 90.000,E1 95.277} C_DIS
LIN {X -0.002,Y -485.338,Z 291.305,A 0.000,B 0.000,C 90.000,E1 90.974} C_DIS
LIN {X -0.177,Y -485.534,Z 291.304,A 0.000,B 0.000,C 90.000,E1 90.688} C_DIS
LIN {X 0.030,Y -486.333,Z 291.282,A 0.000,B 0.000,C 90.000,E1 86.674} C_DIS
LIN {X 0.164,Y -486.285,Z 291.278,A 0.000,B 0.000,C 90.000,E1 86.045} C_DIS
LIN {X -0.116,Y -484.694,Z 291.254,A 0.000,B 0.000,C 90.000,E1 81.781} C_DIS
LIN {X 0.232,Y -484.565,Z 291.253,A 0.000,B 0.000,C 90.000,E1 81.432} C_DIS
LIN {X 0.101,Y -480.503,Z 291.227,A 0.000,B 0.000,C 90.000,E1 76.825} C_DIS
LIN {X -0.002,Y -474.256,Z 291.201,A 0.000,B 0.000,C 90.000,E1 72.181} C_DIS
LIN {X -0.062,Y -473.556,Z 291.199,A 0.000,B 0.000,C 90.000,E1 71.764} C_DIS
LIN {X -0.102,Y -473.555,Z 291.199,A 0.000,B 0.000,C 90.000,E1 71.764} C_DIS
LIN {X -0.073,Y -477.903,Z 291.189,A 0.000,B 0.000,C 90.000,E1 70.007} C_DIS
LIN {X -0.136,Y -484.395,Z 291.175,A 0.000,B 0.000,C 90.000,E1 67.539} C_DIS
LIN {X 0.164,Y -490.249,Z 291.163,A 0.000,B 0.000,C 90.000,E1 65.357} C_DIS
LIN {X -0.110,Y -495.331,Z 291.153,A 0.000,B 0.000,C 90.000,E1 63.563} C_DIS
LIN {X 0.070,Y -502.259,Z 291.140,A 0.000,B 0.000,C 90.000,E1 61.129} C_DIS
LIN {X 0.102,Y -507.482,Z 291.130,A 0.000,B 0.000,C 90.000,E1 59.331} C_DIS
LIN {X -0.182,Y -512.726,Z 291.120,A 0.000,B 0.000,C 90.000,E1 57.582} C_DIS
LIN {X 0.067,Y -516.135,Z 291.113,A 0.000,B 0.000,C 90.000,E1 56.373} C_DIS
LIN {X 0.164,Y -520.280,Z 291.105,A 0.000,B 0.000,C 90.000,E1 54.895} C_DIS
LIN {X -0.035,Y -523.427,Z 291.099,A 0.000,B 0.000,C 90.000,E1 53.749} C_DIS
LIN {X 0.267,Y -525.652,Z 291.094,A 0.000,B 0.000,C 90.000,E1 52.844} C_DIS
LIN {X 0.114,Y -529.054,Z 291.086,A 0.000,B 0.000,C 90.000,E1 51.412} C_DIS
LIN {X -0.066,Y -532.092,Z 291.078,A 0.000,B 0.000,C 90.000,E1 49.989} C_DIS
LIN {X -0.168,Y -533.775,Z 291.073,A 0.000,B 0.000,C 90.000,E1 49.138} C_DIS
LIN {X -0.255,Y -535.715,Z 291.067,A 0.000,B 0.000,C 90.000,E1 48.000} C_DIS
LIN {X 0.079,Y -537.026,Z 291.062,A 0.000,B 0.000,C 90.000,E1 47.106} C_DIS
LIN {X 0.001,Y -538.459,Z 291.055,A 0.000,B 0.000,C 90.000,E1 45.972} C_DIS
LIN {X -0.048,Y -539.571,Z 291.049,A 0.000,B 0.000,C 90.000,E1 44.838} C_DIS
LIN {X -0.085,Y -540.349,Z 291.043,A 0.000,B 0.000,C 90.000,E1 43.704} C_DIS
LIN {X 0.279,Y -540.902,Z 291.036,A 0.000,B 0.000,C 90.000,E1 42.528} C_DIS
LIN {X 0.274,Y -541.190,Z 291.032,A 0.000,B 0.000,C 90.000,E1 41.676} C_DIS
LIN {X -0.083,Y -541.345,Z 291.027,A 0.000,B 0.000,C 90.000,E1 40.862} C_DIS
LIN {X -0.064,Y -541.348,Z 291.021,A 0.000,B 0.000,C 90.000,E1 39.725} C_DIS
LIN {X -0.034,Y -540.922,Z 291.013,A 0.000,B 0.000,C 90.000,E1 38.302} C_DIS
LIN {X 0.054,Y -540.321,Z 291.007,A 0.000,B 0.000,C 90.000,E1 37.156} C_DIS
LIN {X 0.134,Y -539.578,Z 291.000,A 0.000,B 0.000,C 90.000,E1 36.011} C_DIS
LIN {X -0.098,Y -538.400,Z 290.992,A 0.000,B 0.000,C 90.000,E1 34.612} C_DIS
LIN {X 0.096,Y -537.066,Z 290.984,A 0.000,B 0.000,C 90.000,E1 33.166} C_DIS
LIN {X -0.024,Y -535.704,Z 290.976,A 0.000,B 0.000,C 90.000,E1 31.750} C_DIS
LIN {X 0.274,Y -533.903,Z 290.967,A 0.000,B 0.000,C 90.000,E1 30.001} C_DIS
LIN {X 0.001,Y -532.086,Z 290.957,A 0.000,B 0.000,C 90.000,E1 28.309} C_DIS
LIN {X 0.275,Y -530.896,Z 290.951,A 0.000,B 0.000,C 90.000,E1 27.129} C_DIS
LIN {X -0.131,Y -528.750,Z 290.940,A 0.000,B 0.000,C 90.000,E1 25.155} C_DIS
LIN {X 0.192,Y -527.067,Z 290.930,A 0.000,B 0.000,C 90.000,E1 23.387} C_DIS
LIN {X -0.255,Y -525.261,Z 290.919,A 0.000,B 0.000,C 90.000,E1 21.408} C_DIS
LIN {X -0.279,Y -523.478,Z 290.906,A 0.000,B 0.000,C 90.000,E1 19.087} C_DIS
LIN {X -0.185,Y -522.031,Z 290.895,A 0.000,B 0.000,C 90.000,E1 17.040} C_DIS
LIN {X -0.157,Y -520.475,Z 290.878,A 0.000,B 0.000,C 90.000,E1 14.120} C_DIS
LIN {X -0.049,Y -519.785,Z 290.869,A 0.000,B 0.000,C 90.000,E1 12.355} C_DIS
LIN {X -0.081,Y -519.079,Z 290.854,A 0.000,B 0.000,C 90.000,E1 9.726} C_DIS
LIN {X 0.230,Y -518.863,Z 290.844,A 0.000,B 0.000,C 90.000,E1 7.936} C_DIS
LIN {X -0.141,Y -519.036,Z 290.828,A 0.000,B 0.000,C 90.000,E1 5.049} C_DIS
LIN {X 0.081,Y -519.450,Z 290.818,A 0.000,B 0.000,C 90.000,E1 3.269} C_DIS
LIN {X -0.173,Y -519.983,Z 290.810,A 0.000,B 0.000,C 90.000,E1 1.835} C_DIS
LIN {X 0.049,Y -521.571,Z 290.794,A 0.000,B 0.000,C 90.000,E1 358.912} C_DIS
LIN {X -0.267,Y -523.147,Z 290.783,A 0.000,B 0.000,C 90.000,E1 356.906} C_DIS
LIN {X 0.087,Y -524.759,Z 290.773,A 0.000,B 0.000,C 90.000,E1 355.122} C_DIS
LIN {X -0.021,Y -531.852,Z 290.744,A 0.000,B 0.000,C 90.000,E1 349.926} C_DIS
LIN {X -0.221,Y -535.986,Z 290.733,A 0.000,B 0.000,C 90.000,E1 347.937} C_DIS
LIN {X -0.193,Y -540.843,Z 290.722,A 0.000,B 0.000,C 90.000,E1 345.936} C_DIS
LIN {X 0.094,Y -545.830,Z 290.711,A 0.000,B 0.000,C 90.000,E1 343.921} C_DIS
LIN {X 0.133,Y -551.174,Z 290.700,A 0.000,B 0.000,C 90.000,E1 341.945} C_DIS
LIN {X -0.102,Y -560.461,Z 290.683,A 0.000,B 0.000,C 90.000,E1 338.901} C_DIS
LIN {X 0.023,Y -565.942,Z 290.674,A 0.000,B 0.000,C 90.000,E1 337.230} C_DIS
LIN {X 0.324,Y -569.664,Z 290.667,A 0.000,B 0.000,C 90.000,E1 336.102} C_DIS
LIN {X -0.247,Y -574.395,Z 290.660,A 0.000,B 0.000,C 90.000,E1 334.793} C_DIS
LIN {X 0.129,Y -580.253,Z 290.651,A 0.000,B 0.000,C 90.000,E1 333.127} C_DIS
LIN {X 0.243,Y -584.995,Z 290.643,A 0.000,B 0.000,C 90.000,E1 331.769} C_DIS
LIN {X -0.079,Y -589.577,Z 290.636,A 0.000,B 0.000,C 90.000,E1 330.461} C_DIS
LIN {X -0.030,Y -594.050,Z 290.629,A 0.000,B 0.000,C 90.000,E1 329.125} C_DIS
LIN {X 0.101,Y -598.590,Z 290.621,A 0.000,B 0.000,C 90.000,E1 327.788} C_DIS
LIN {X 0.044,Y -604.114,Z 290.612,A 0.000,B 0.000,C 90.000,E1 326.215} C_DIS
LIN {X 0.169,Y -608.962,Z 290.605,A 0.000,B 0.000,C 90.000,E1 324.895} C_DIS
LIN {X -0.124,Y -613.688,Z 290.598,A 0.000,B 0.000,C 90.000,E1 323.623} C_DIS
LIN {X 0.213,Y -617.268,Z 290.592,A 0.000,B 0.000,C 90.000,E1 322.557} C_DIS
LIN {X 0.108,Y -620.658,Z 290.586,A 0.000,B 0.000,C 90.000,E1 321.537} C_DIS
LIN {X 0.227,Y -625.498,Z 290.578,A 0.000,B 0.000,C 90.000,E1 319.989} C_DIS
LIN {X 0.086,Y -629.351,Z 290.571,A 0.000,B 0.000,C 90.000,E1 318.728} C_DIS
LIN {X 0.064,Y -632.260,Z 290.565,A 0.000,B 0.000,C 90.000,E1 317.715} C_DIS
LIN {X -0.121,Y -636.595,Z 290.557,A 0.000,B 0.000,C 90.000,E1 316.215} C_DIS
LIN {X 0.315,Y -640.228,Z 290.550,A 0.000,B 0.000,C 90.000,E1 314.919} C_DIS
LIN {X -0.094,Y -643.805,Z 290.543,A 0.000,B 0.000,C 90.000,E1 313.704} C_DIS
LIN {X 0.084,Y -646.530,Z 290.537,A 0.000,B 0.000,C 90.000,E1 312.690} C_DIS
LIN {X 0.299,Y -649.115,Z 290.532,A 0.000,B 0.000,C 90.000,E1 311.676} C_DIS
LIN {X 0.059,Y -651.993,Z 290.525,A 0.000,B 0.000,C 90.000,E1 310.458} C_DIS
LIN {X -0.087,Y -654.112,Z 290.519,A 0.000,B 0.000,C 90.000,E1 309.483} C_DIS
LIN {X -0.159,Y -656.403,Z 290.513,A 0.000,B 0.000,C 90.000,E1 308.257} C_DIS
LIN {X -0.204,Y -657.607,Z 290.508,A 0.000,B 0.000,C 90.000,E1 307.523} C_DIS
LIN {X 0.231,Y -659.009,Z 290.503,A 0.000,B 0.000,C 90.000,E1 306.503} C_DIS
LIN {X -0.186,Y -659.876,Z 290.499,A 0.000,B 0.000,C 90.000,E1 305.804} C_DIS
LIN {X -0.152,Y -660.255,Z 290.496,A 0.000,B 0.000,C 90.000,E1 305.311} C_DIS
LIN {X -0.011,Y -660.562,Z 290.492,A 0.000,B 0.000,C 90.000,E1 304.565} C_DIS
LIN {X -0.370,Y -660.814,Z 290.485,A 0.000,B 0.000,C 90.000,E1 303.372} C_DIS
LIN {X -0.216,Y -660.615,Z 290.481,A 0.000,B 0.000,C 90.000,E1 302.625} C_DIS
LIN {X -0.185,Y -660.388,Z 290.478,A 0.000,B 0.000,C 90.000,E1 302.133} C_DIS
LIN {X -0.041,Y -659.673,Z 290.474,A 0.000,B 0.000,C 90.000,E1 301.386} C_DIS
LIN {X -0.244,Y -658.644,Z 290.470,A 0.000,B 0.000,C 90.000,E1 300.669} C_DIS
LIN {X -0.121,Y -657.311,Z 290.466,A 0.000,B 0.000,C 90.000,E1 299.922} C_DIS
LIN {X -0.227,Y -655.193,Z 290.461,A 0.000,B 0.000,C 90.000,E1 298.949} C_DIS
LIN {X -0.138,Y -651.657,Z 290.453,A 0.000,B 0.000,C 90.000,E1 297.462} C_DIS
LIN {X -0.216,Y -648.556,Z 290.446,A 0.000,B 0.000,C 90.000,E1 296.232} C_DIS
LIN {X 0.114,Y -643.907,Z 290.436,A 0.000,B 0.000,C 90.000,E1 294.463} C_DIS
LIN {X 0.075,Y -639.162,Z 290.426,A 0.000,B 0.000,C 90.000,E1 292.717} C_DIS
LIN {X -0.277,Y -633.905,Z 290.415,A 0.000,B 0.000,C 90.000,E1 290.737} C_DIS
LIN {X 0.192,Y -628.811,Z 290.404,A 0.000,B 0.000,C 90.000,E1 288.671} C_DIS
LIN {X -0.066,Y -624.622,Z 290.394,A 0.000,B 0.000,C 90.000,E1 286.913} C_DIS
LIN {X 0.136,Y -619.854,Z 290.381,A 0.000,B 0.000,C 90.000,E1 284.592} C_DIS
LIN {X 0.152,Y -614.236,Z 290.363,A 0.000,B 0.000,C 90.000,E1 281.243} C_DIS
LIN {X -0.147,Y -610.921,Z 290.348,A 0.000,B 0.000,C 90.000,E1 278.681} C_DIS
LIN {X 0.121,Y -608.383,Z 290.332,A 0.000,B 0.000,C 90.000,E1 275.796} C_DIS
LIN {X 0.189,Y -606.908,Z 290.316,A 0.000,B 0.000,C 90.000,E1 272.922} C_DIS
LIN {X -0.071,Y -606.475,Z 290.305,A 0.000,B 0.000,C 90.000,E1 270.859} C_DIS
LIN {X 0.260,Y -606.631,Z 290.293,A 0.000,B 0.000,C 90.000,E1 268.740} C_DIS
LIN {X 0.188,Y -608.196,Z 290.274,A 0.000,B 0.000,C 90.000,E1 265.355} C_DIS
LIN {X -0.221,Y -609.670,Z 290.264,A 0.000,B 0.000,C 90.000,E1 263.571} C_DIS
LIN {X 0.163,Y -612.163,Z 290.251,A 0.000,B 0.000,C 90.000,E1 261.197} C_DIS
LIN {X -0.108,Y -615.718,Z 290.237,A 0.000,B 0.000,C 90.000,E1 258.634} C_DIS
LIN {X -0.069,Y -618.454,Z 290.227,A 0.000,B 0.000,C 90.000,E1 256.825} C_DIS
LIN {X 0.153,Y -620.412,Z 290.220,A 0.000,B 0.000,C 90.000,E1 255.519} C_DIS
LIN {X -0.131,Y -621.960,Z 290.214,A 0.000,B 0.000,C 90.000,E1 254.519} C_DIS
LIN {X -0.016,Y -622.880,Z 290.210,A 0.000,B 0.000,C 90.000,E1 253.740} C_DIS
LIN {X -0.105,Y -623.792,Z 290.204,A 0.000,B 0.000,C 90.000,E1 252.725} C_DIS
LIN {X 0.167,Y -624.899,Z 290.195,A 0.000,B 0.000,C 90.000,E1 251.167} C_DIS
LIN {X -0.078,Y -625.170,Z 290.191,A 0.000,B 0.000,C 90.000,E1 250.423} C_DIS
LIN {X 0.057,Y -625.256,Z 290.186,A 0.000,B 0.000,C 90.000,E1 249.390} C_DIS
LIN {X -0.170,Y -625.005,Z 290.181,A 0.000,B 0.000,C 90.000,E1 248.646} C_DIS
LIN {X 0.184,Y -624.545,Z 290.177,A 0.000,B 0.000,C 90.000,E1 247.847} C_DIS
LIN {X -0.045,Y -623.886,Z 290.173,A 0.000,B 0.000,C 90.000,E1 247.102} C_DIS
LIN {X -0.282,Y -622.935,Z 290.169,A 0.000,B 0.000,C 90.000,E1 246.357} C_DIS
LIN {X 0.033,Y -621.382,Z 290.163,A 0.000,B 0.000,C 90.000,E1 245.305} C_DIS
LIN {X 0.024,Y -619.949,Z 290.159,A 0.000,B 0.000,C 90.000,E1 244.537} C_DIS
LIN {X 0.005,Y -618.267,Z 290.154,A 0.000,B 0.000,C 90.000,E1 243.768} C_DIS
LIN {X -0.045,Y -615.830,Z 290.149,A 0.000,B 0.000,C 90.000,E1 242.743} C_DIS
LIN {X 0.130,Y -612.445,Z 290.141,A 0.000,B 0.000,C 90.000,E1 241.435} C_DIS
LIN {X -0.010,Y -609.577,Z 290.136,A 0.000,B 0.000,C 90.000,E1 240.411} C_DIS
LIN {X -0.112,Y -606.620,Z 290.130,A 0.000,B 0.000,C 90.000,E1 239.380} C_DIS
LIN {X -0.037,Y -603.579,Z 290.124,A 0.000,B 0.000,C 90.000,E1 238.329} C_DIS
LIN {X -0.283,Y -599.694,Z 290.117,A 0.000,B 0.000,C 90.000,E1 237.041} C_DIS
LIN {X 0.228,Y -595.636,Z 290.109,A 0.000,B 0.000,C 90.000,E1 235.674} C_DIS
LIN {X -0.049,Y -592.230,Z 290.104,A 0.000,B 0.000,C 90.000,E1 234.642} C_DIS
LIN {X -0.098,Y -586.932,Z 290.095,A 0.000,B 0.000,C 90.000,E1 233.050} C_DIS
LIN {X -0.243,Y -581.944,Z 290.086,A 0.000,B 0.000,C 90.000,E1 231.457} C_DIS
LIN {X -0.006,Y -578.555,Z 290.080,A 0.000,B 0.000,C 90.000,E1 230.356} C_DIS
LIN {X -0.054,Y -570.955,Z 290.066,A 0.000,B 0.000,C 90.000,E1 227.919} C_DIS
LIN {X 0.076,Y -566.779,Z 290.059,A 0.000,B 0.000,C 90.000,E1 226.539} C_DIS
LIN {X -0.214,Y -561.620,Z 290.049,A 0.000,B 0.000,C 90.000,E1 224.919} C_DIS
LIN {X 0.063,Y -558.231,Z 290.043,A 0.000,B 0.000,C 90.000,E1 223.785} C_DIS
LIN {X -0.008,Y -553.133,Z 290.034,A 0.000,B 0.000,C 90.000,E1 222.123} C_DIS
LIN {X -0.101,Y -547.132,Z 290.023,A 0.000,B 0.000,C 90.000,E1 220.172} C_DIS
LIN {X 0.054,Y -541.962,Z 290.014,A 0.000,B 0.000,C 90.000,E1 218.463} C_DIS
LIN {X 0.172,Y -537.699,Z 290.006,A 0.000,B 0.000,C 90.000,E1 217.030} C_DIS
LIN {X 0.206,Y -531.763,Z 289.995,A 0.000,B 0.000,C 90.000,E1 215.025} C_DIS
LIN {X -0.082,Y -525.944,Z 289.984,A 0.000,B 0.000,C 90.000,E1 213.038} C_DIS
LIN {X -0.130,Y -519.752,Z 289.971,A 0.000,B 0.000,C 90.000,E1 210.718} C_DIS
LIN {X 0.105,Y -513.032,Z 289.956,A 0.000,B 0.000,C 90.000,E1 208.052} C_DIS
LIN {X -0.102,Y -506.773,Z 289.941,A 0.000,B 0.000,C 90.000,E1 205.412} C_DIS
LIN {X -0.112,Y -501.653,Z 289.928,A 0.000,B 0.000,C 90.000,E1 203.025} C_DIS
LIN {X -0.137,Y -498.019,Z 289.918,A 0.000,B 0.000,C 90.000,E1 201.227} C_DIS
LIN {X 0.040,Y -494.556,Z 289.908,A 0.000,B 0.000,C 90.000,E1 199.396} C_DIS
LIN {X -0.110,Y -490.358,Z 289.894,A 0.000,B 0.000,C 90.000,E1 196.985} C_DIS
LIN {X -0.060,Y -486.482,Z 289.881,A 0.000,B 0.000,C 90.000,E1 194.537} C_DIS
LIN {X -0.118,Y -483.788,Z 289.871,A 0.000,B 0.000,C 90.000,E1 192.703} C_DIS
LIN {X -0.112,Y -480.931,Z 289.859,A 0.000,B 0.000,C 90.000,E1 190.546} C_DIS
LIN {X -0.254,Y -478.297,Z 289.847,A 0.000,B 0.000,C 90.000,E1 188.398} C_DIS
LIN {X 0.159,Y -476.235,Z 289.836,A 0.000,B 0.000,C 90.000,E1 186.486} C_DIS
LIN {X -0.144,Y -474.998,Z 289.829,A 0.000,B 0.000,C 90.000,E1 185.277} C_DIS
LIN {X 0.108,Y -472.660,Z 289.815,A 0.000,B 0.000,C 90.000,E1 182.751} C_DIS
LIN {X 0.000,Y -470.892,Z 289.803,A 0.000,B 0.000,C 90.000,E1 180.573} C_DIS
LIN {X 0.097,Y -469.442,Z 289.789,A 0.000,B 0.000,C 90.000,E1 178.051} C_DIS
LIN {X -0.047,Y -468.044,Z 289.770,A 0.000,B 0.000,C 90.000,E1 174.609} C_DIS
LIN {X -0.121,Y -467.665,Z 289.758,A 0.000,B 0.000,C 90.000,E1 172.413} C_DIS
LIN {X -0.043,Y -467.340,Z 289.742,A 0.000,B 0.000,C 90.000,E1 169.567} C_DIS
LIN {X 0.009,Y -467.651,Z 289.725,A 0.000,B 0.000,C 90.000,E1 166.408} C_DIS
LIN {X -0.121,Y -469.005,Z 289.705,A 0.000,B 0.000,C 90.000,E1 162.960} C_DIS
LIN {X -0.181,Y -471.032,Z 289.688,A 0.000,B 0.000,C 90.000,E1 159.826} C_DIS
LIN {X 0.055,Y -472.286,Z 289.679,A 0.000,B 0.000,C 90.000,E1 158.230} C_DIS
LIN {X 0.129,Y -475.097,Z 289.664,A 0.000,B 0.000,C 90.000,E1 155.409} C_DIS
LIN {X 0.049,Y -478.861,Z 289.646,A 0.000,B 0.000,C 90.000,E1 152.308} C_DIS
LIN {X 0.171,Y -482.138,Z 289.634,A 0.000,B 0.000,C 90.000,E1 150.127} C_DIS
LIN {X 0.203,Y -486.190,Z 289.621,A 0.000,B 0.000,C 90.000,E1 147.661} C_DIS
LIN {X -0.051,Y -489.910,Z 289.609,A 0.000,B 0.000,C 90.000,E1 145.548} C_DIS
LIN {X 0.244,Y -492.586,Z 289.600,A 0.000,B 0.000,C 90.000,E1 143.989} C_DIS
LIN {X 0.059,Y -495.716,Z 289.590,A 0.000,B 0.000,C 90.000,E1 142.190} C_DIS
LIN {X -0.183,Y -497.719,Z 289.583,A 0.000,B 0.000,C 90.000,E1 141.009} C_DIS
LIN {X -0.015,Y -499.519,Z 289.577,A 0.000,B 0.000,C 90.000,E1 139.784} C_DIS
LIN {X 0.114,Y -501.182,Z 289.570,A 0.000,B 0.000,C 90.000,E1 138.566} C_DIS
LIN {X 0.024,Y -502.161,Z 289.565,A 0.000,B 0.000,C 90.000,E1 137.676} C_DIS
LIN {X -0.021,Y -502.986,Z 289.560,A 0.000,B 0.000,C 90.000,E1 136.782} C_DIS
LIN {X -0.083,Y -503.487,Z 289.555,A 0.000,B 0.000,C 90.000,E1 135.891} C_DIS
LIN {X -0.135,Y -503.785,Z 289.550,A 0.000,B 0.000,C 90.000,E1 135.000} C_DIS
LIN {X 0.037,Y -503.801,Z 289.543,A 0.000,B 0.000,C 90.000,E1 133.785} C_DIS
LIN {X -0.019,Y -503.469,Z 289.538,A 0.000,B 0.000,C 90.000,E1 132.894} C_DIS
LIN {X -0.049,Y -502.937,Z 289.533,A 0.000,B 0.000,C 90.000,E1 132.000} C_DIS
LIN {X 0.133,Y -501.815,Z 289.527,A 0.000,B 0.000,C 90.000,E1 130.782} C_DIS
LIN {X 0.097,Y -500.798,Z 289.522,A 0.000,B 0.000,C 90.000,E1 129.886} C_DIS
LIN {X 0.049,Y -499.626,Z 289.517,A 0.000,B 0.000,C 90.000,E1 128.991} C_DIS
LIN {X -0.271,Y -497.530,Z 289.508,A 0.000,B 0.000,C 90.000,E1 127.523} C_DIS
LIN {X -0.103,Y -495.696,Z 289.502,A 0.000,B 0.000,C 90.000,E1 126.297} C_DIS
LIN {X -0.257,Y -493.662,Z 289.495,A 0.000,B 0.000,C 90.000,E1 125.105} C_DIS
LIN {X -0.033,Y -491.429,Z 289.488,A 0.000,B 0.000,C 90.000,E1 123.865} C_DIS
LIN {X 0.235,Y -487.977,Z 289.478,A 0.000,B 0.000,C 90.000,E1 122.005} C_DIS
LIN {X -0.094,Y -484.505,Z 289.468,A 0.000,B 0.000,C 90.000,E1 120.207} C_DIS
LIN {X 0.127,Y -480.298,Z 289.456,A 0.000,B 0.000,C 90.000,E1 118.025} C_DIS
LIN {X 0.039,Y -477.313,Z 289.447,A 0.000,B 0.000,C 90.000,E1 116.488} C_DIS
LIN {X -0.278,Y -474.826,Z 289.440,A 0.000,B 0.000,C 90.000,E1 115.283} C_DIS
LIN {X -0.007,Y -472.518,Z 289.433,A 0.000,B 0.000,C 90.000,E1 114.003} C_DIS
LIN {X -0.288,Y -468.378,Z 289.421,A 0.000,B 0.000,C 90.000,E1 111.844} C_DIS
LIN {X -0.171,Y -465.008,Z 289.411,A 0.000,B 0.000,C 90.000,E1 109.939} C_DIS
LIN {X 0.220,Y -461.269,Z 289.398,A 0.000,B 0.000,C 90.000,E1 107.692} C_DIS
LIN {X 0.181,Y -461.277,Z 289.398,A 0.000,B 0.000,C 90.000,E1 107.692} C_DIS
LIN {X 0.150,Y -467.870,Z 289.383,A 0.000,B 0.000,C 90.000,E1 104.828} C_DIS
LIN {X 0.178,Y -475.430,Z 289.358,A 0.000,B 0.000,C 90.000,E1 100.433} C_DIS
LIN {X 0.016,Y -476.081,Z 289.356,A 0.000,B 0.000,C 90.000,E1 100.141} C_DIS
LIN {X -0.180,Y -482.004,Z 289.331,A 0.000,B 0.000,C 90.000,E1 95.511} C_DIS
LIN {X -0.199,Y -482.514,Z 289.325,A 0.000,B 0.000,C 90.000,E1 94.588} C_DIS
LIN {X 0.090,Y -485.449,Z 289.305,A 0.000,B 0.000,C 90.000,E1 90.859} C_DIS
LIN {X 0.228,Y -485.505,Z 289.301,A 0.000,B 0.000,C 90.000,E1 90.229} C_DIS
LIN {X 0.123,Y -486.381,Z 289.281,A 0.000,B 0.000,C 90.000,E1 86.560} C_DIS
LIN {X -0.052,Y -486.365,Z 289.279,A 0.000,B 0.000,C 90.000,E1 86.274} C_DIS
LIN {X 0.037,Y -484.690,Z 289.254,A 0.000,B 0.000,C 90.000,E1 81.659} C_DIS
LIN {X 0.182,Y -484.073,Z 289.250,A 0.000,B 0.000,C 90.000,E1 81.027} C_DIS
LIN {X -0.162,Y -480.640,Z 289.228,A 0.000,B 0.000,C 90.000,E1 77.061} C_DIS
LIN {X -0.196,Y -480.345,Z 289.226,A 0.000,B 0.000,C 90.000,E1 76.756} C_DIS
LIN {X 0.175,Y -474.153,Z 289.200,A 0.000,B 0.000,C 90.000,E1 72.054} C_DIS
LIN {X 0.041,Y -473.210,Z 289.198,A 0.000,B 0.000,C 90.000,E1 71.583} C_DIS
LIN {X 0.002,Y -473.208,Z 289.198,A 0.000,B 0.000,C 90.000,E1 71.583} C_DIS
LIN {X 0.101,Y -477.386,Z 289.188,A 0.000,B 0.000,C 90.000,E1 69.880} C_DIS
LIN {X 0.030,Y -483.911,Z 289.175,A 0.000,B 0.000,C 90.000,E1 67.411} C_DIS
LIN {X -0.125,Y -489.728,Z 289.163,A 0.000,B 0.000,C 90.000,E1 65.281} C_DIS
LIN {X -0.218,Y -493.989,Z 289.154,A 0.000,B 0.000,C 90.000,E1 63.768} C_DIS
LIN {X 0.153,Y -500.891,Z 289.141,A 0.000,B 0.000,C 90.000,E1 61.307} C_DIS
LIN {X 0.222,Y -506.984,Z 289.129,A 0.000,B 0.000,C 90.000,E1 59.203} C_DIS
LIN {X -0.165,Y -513.097,Z 289.118,A 0.000,B 0.000,C 90.000,E1 57.168} C_DIS
LIN {X 0.016,Y -517.290,Z 289.109,A 0.000,B 0.000,C 90.000,E1 55.674} C_DIS
LIN {X 0.192,Y -520.606,Z 289.103,A 0.000,B 0.000,C 90.000,E1 54.482} C_DIS
LIN {X -0.004,Y -523.641,Z 289.096,A 0.000,B 0.000,C 90.000,E1 53.336} C_DIS
LIN {X -0.158,Y -526.454,Z 289.090,A 0.000,B 0.000,C 90.000,E1 52.190} C_DIS
LIN {X 0.080,Y -528.444,Z 289.085,A 0.000,B 0.000,C 90.000,E1 51.295} C_DIS
LIN {X 0.309,Y -531.490,Z 289.077,A 0.000,B 0.000,C 90.000,E1 49.828} C_DIS
LIN {X 0.190,Y -533.670,Z 289.071,A 0.000,B 0.000,C 90.000,E1 48.690} C_DIS
LIN {X -0.308,Y -535.931,Z 289.063,A 0.000,B 0.000,C 90.000,E1 47.310} C_DIS
LIN {X -0.009,Y -537.385,Z 289.056,A 0.000,B 0.000,C 90.000,E1 46.134} C_DIS
LIN {X -0.059,Y -538.274,Z 289.052,A 0.000,B 0.000,C 90.000,E1 45.283} C_DIS
LIN {X -0.101,Y -538.985,Z 289.047,A 0.000,B 0.000,C 90.000,E1 44.433} C_DIS
LIN {X 0.245,Y -539.536,Z 289.042,A 0.000,B 0.000,C 90.000,E1 43.542} C_DIS
LIN {X 0.226,Y -539.952,Z 289.037,A 0.000,B 0.000,C 90.000,E1 42.690} C_DIS
LIN {X -0.181,Y -540.297,Z 289.031,A 0.000,B 0.000,C 90.000,E1 41.595} C_DIS
LIN {X -0.182,Y -540.444,Z 289.025,A 0.000,B 0.000,C 90.000,E1 40.458} C_DIS
LIN {X 0.215,Y -540.416,Z 289.020,A 0.000,B 0.000,C 90.000,E1 39.564} C_DIS
LIN {X -0.129,Y -540.025,Z 289.014,A 0.000,B 0.000,C 90.000,E1 38.463} C_DIS
LIN {X -0.070,Y -539.614,Z 289.009,A 0.000,B 0.000,C 90.000,E1 37.604} C_DIS
LIN {X 0.005,Y -538.896,Z 289.003,A 0.000,B 0.000,C 90.000,E1 36.457} C_DIS
LIN {X 0.066,Y -538.027,Z 288.996,A 0.000,B 0.000,C 90.000,E1 35.311} C_DIS
LIN {X -0.199,Y -537.001,Z 288.990,A 0.000,B 0.000,C 90.000,E1 34.199} C_DIS
LIN {X -0.035,Y -535.394,Z 288.980,A 0.000,B 0.000,C 90.000,E1 32.467} C_DIS
LIN {X -0.023,Y -533.591,Z 288.971,A 0.000,B 0.000,C 90.000,E1 30.747} C_DIS
LIN {X -0.039,Y -531.773,Z 288.961,A 0.000,B 0.000,C 90.000,E1 29.027} C_DIS
LIN {X -0.110,Y -529.929,Z 288.952,A 0.000,B 0.000,C 90.000,E1 27.308} C_DIS
LIN {X -0.244,Y -528.017,Z 288.942,A 0.000,B 0.000,C 90.000,E1 25.591} C_DIS
LIN {X 0.061,Y -526.325,Z 288.932,A 0.000,B 0.000,C 90.000,E1 23.823} C_DIS
LIN {X 0.082,Y -524.438,Z 288.921,A 0.000,B 0.000,C 90.000,E1 21.791} C_DIS
LIN {X -0.289,Y -522.365,Z 288.907,A 0.000,B 0.000,C 90.000,E1 19.214} C_DIS
LIN {X -0.062,Y -520.896,Z 288.895,A 0.000,B 0.000,C 90.000,E1 17.149} C_DIS
LIN {X -0.214,Y -519.364,Z 288.881,A 0.000,B 0.000,C 90.000,E1 14.537} C_DIS
LIN {X -0.132,Y -518.529,Z 288.869,A 0.000,B 0.000,C 90.000,E1 12.479} C_DIS
LIN {X -0.191,Y -517.736,Z 288.855,A 0.000,B 0.000,C 90.000,E1 9.849} C_DIS
LIN {X 0.157,Y -517.445,Z 288.843,A 0.000,B 0.000,C 90.000,E1 7.757} C_DIS
LIN {X -0.182,Y -517.544,Z 288.830,A 0.000,B 0.000,C 90.000,E1 5.448} C_DIS
LIN {X -0.003,Y -517.931,Z 288.820,A 0.000,B 0.000,C 90.000,E1 3.669} C_DIS
LIN {X -0.053,Y -519.006,Z 288.804,A 0.000,B 0.000,C 90.000,E1 0.745} C_DIS
LIN {X -0.112,Y -520.730,Z 288.789,A 0.000,B 0.000,C 90.000,E1 358.051} C_DIS
LIN {X 0.073,Y -522.434,Z 288.778,A 0.000,B 0.000,C 90.000,E1 355.988} C_DIS
LIN {X -0.206,Y -525.491,Z 288.762,A 0.000,B 0.000,C 90.000,E1 353.109} C_DIS
LIN {X -0.016,Y -533.182,Z 288.736,A 0.000,B 0.000,C 90.000,E1 348.465} C_DIS
LIN {X 0.065,Y -539.396,Z 288.722,A 0.000,B 0.000,C 90.000,E1 345.880} C_DIS
LIN {X -0.211,Y -544.393,Z 288.711,A 0.000,B 0.000,C 90.000,E1 343.921} C_DIS
LIN {X 0.133,Y -551.347,Z 288.697,A 0.000,B 0.000,C 90.000,E1 341.348} C_DIS
LIN {X -0.113,Y -561.823,Z 288.678,A 0.000,B 0.000,C 90.000,E1 338.028} C_DIS
LIN {X 0.044,Y -567.392,Z 288.669,A 0.000,B 0.000,C 90.000,E1 336.357} C_DIS
LIN {X 0.026,Y -573.055,Z 288.660,A 0.000,B 0.000,C 90.000,E1 334.717} C_DIS
LIN {X 0.121,Y -578.961,Z 288.651,A 0.000,B 0.000,C 90.000,E1 333.076} C_DIS
LIN {X 0.073,Y -584.635,Z 288.642,A 0.000,B 0.000,C 90.000,E1 331.463} C_DIS
LIN {X 0.146,Y -588.352,Z 288.636,A 0.000,B 0.000,C 90.000,E1 330.383} C_DIS
LIN {X -0.030,Y -594.625,Z 288.625,A 0.000,B 0.000,C 90.000,E1 328.535} C_DIS
LIN {X -0.265,Y -601.070,Z 288.615,A 0.000,B 0.000,C 90.000,E1 326.707} C_DIS
LIN {X -0.022,Y -607.774,Z 288.605,A 0.000,B 0.000,C 90.000,E1 324.848} C_DIS
LIN {X 0.021,Y -612.520,Z 288.598,A 0.000,B 0.000,C 90.000,E1 323.543} C_DIS
LIN {X 0.345,Y -616.118,Z 288.592,A 0.000,B 0.000,C 90.000,E1 322.477} C_DIS
LIN {X 0.227,Y -619.553,Z 288.586,A 0.000,B 0.000,C 90.000,E1 321.457} C_DIS
LIN {X 0.327,Y -624.447,Z 288.577,A 0.000,B 0.000,C 90.000,E1 319.908} C_DIS
LIN {X -0.302,Y -628.309,Z 288.570,A 0.000,B 0.000,C 90.000,E1 318.690} C_DIS
LIN {X 0.136,Y -631.249,Z 288.565,A 0.000,B 0.000,C 90.000,E1 317.634} C_DIS
LIN {X -0.170,Y -636.320,Z 288.555,A 0.000,B 0.000,C 90.000,E1 315.891} C_DIS
LIN {X 0.262,Y -639.905,Z 288.548,A 0.000,B 0.000,C 90.000,E1 314.595} C_DIS
LIN {X -0.156,Y -643.445,Z 288.541,A 0.000,B 0.000,C 90.000,E1 313.380} C_DIS
LIN {X 0.088,Y -645.467,Z 288.537,A 0.000,B 0.000,C 90.000,E1 312.609} C_DIS
LIN {X 0.288,Y -648.048,Z 288.531,A 0.000,B 0.000,C 90.000,E1 311.595} C_DIS
LIN {X 0.028,Y -650.903,Z 288.524,A 0.000,B 0.000,C 90.000,E1 310.378} C_DIS
LIN {X -0.134,Y -652.968,Z 288.519,A 0.000,B 0.000,C 90.000,E1 309.402} C_DIS
LIN {X 0.232,Y -655.642,Z 288.511,A 0.000,B 0.000,C 90.000,E1 307.890} C_DIS
LIN {X -0.275,Y -657.094,Z 288.505,A 0.000,B 0.000,C 90.000,E1 306.950} C_DIS
LIN {X 0.211,Y -658.064,Z 288.501,A 0.000,B 0.000,C 90.000,E1 306.171} C_DIS
LIN {X -0.299,Y -658.610,Z 288.498,A 0.000,B 0.000,C 90.000,E1 305.724} C_DIS
LIN {X -0.248,Y -659.103,Z 288.493,A 0.000,B 0.000,C 90.000,E1 304.739} C_DIS
LIN {X 0.352,Y -659.305,Z 288.487,A 0.000,B 0.000,C 90.000,E1 303.706} C_DIS
LIN {X -0.064,Y -659.350,Z 288.483,A 0.000,B 0.000,C 90.000,E1 303.007} C_DIS
LIN {X 0.068,Y -659.041,Z 288.479,A 0.000,B 0.000,C 90.000,E1 302.260} C_DIS
LIN {X -0.148,Y -658.404,Z 288.475,A 0.000,B 0.000,C 90.000,E1 301.544} C_DIS
LIN {X -0.022,Y -657.429,Z 288.471,A 0.000,B 0.000,C 90.000,E1 300.797} C_DIS
LIN {X 0.088,Y -656.170,Z 288.467,A 0.000,B 0.000,C 90.000,E1 300.050} C_DIS
LIN {X -0.145,Y -654.651,Z 288.463,A 0.000,B 0.000,C 90.000,E1 299.333} C_DIS
LIN {X 0.184,Y -652.944,Z 288.459,A 0.000,B 0.000,C 90.000,E1 298.565} C_DIS
LIN {X 0.030,Y -650.573,Z 288.453,A 0.000,B 0.000,C 90.000,E1 297.590} C_DIS
LIN {X 0.024,Y -646.836,Z 288.445,A 0.000,B 0.000,C 90.000,E1 296.104} C_DIS
LIN {X 0.238,Y -642.830,Z 288.437,A 0.000,B 0.000,C 90.000,E1 294.591} C_DIS
LIN {X 0.174,Y -638.100,Z 288.427,A 0.000,B 0.000,C 90.000,E1 292.845} C_DIS
LIN {X 0.024,Y -632.820,Z 288.416,A 0.000,B 0.000,C 90.000,E1 290.844} C_DIS
LIN {X 0.240,Y -627.079,Z 288.403,A 0.000,B 0.000,C 90.000,E1 288.544} C_DIS
LIN {X 0.316,Y -622.377,Z 288.392,A 0.000,B 0.000,C 90.000,E1 286.496} C_DIS
LIN {X 0.145,Y -618.711,Z 288.382,A 0.000,B 0.000,C 90.000,E1 284.717} C_DIS
LIN {X -0.116,Y -612.683,Z 288.362,A 0.000,B 0.000,C 90.000,E1 281.130} C_DIS
LIN {X -0.119,Y -609.130,Z 288.346,A 0.000,B 0.000,C 90.000,E1 278.276} C_DIS
LIN {X -0.234,Y -606.926,Z 288.331,A 0.000,B 0.000,C 90.000,E1 275.682} C_DIS
LIN {X -0.214,Y -605.507,Z 288.316,A 0.000,B 0.000,C 90.000,E1 272.808} C_DIS
LIN {X 0.174,Y -605.200,Z 288.307,A 0.000,B 0.000,C 90.000,E1 271.203} C_DIS
LIN {X -0.138,Y -605.277,Z 288.295,A 0.000,B 0.000,C 90.000,E1 269.141} C_DIS
LIN {X 0.257,Y -607.030,Z 288.273,A 0.000,B 0.000,C 90.000,E1 265.184} C_DIS
LIN {X -0.115,Y -608.534,Z 288.263,A 0.000,B 0.000,C 90.000,E1 263.394} C_DIS
LIN {X -0.105,Y -611.422,Z 288.249,A 0.000,B 0.000,C 90.000,E1 260.792} C_DIS
LIN {X 0.079,Y -614.333,Z 288.237,A 0.000,B 0.000,C 90.000,E1 258.701} C_DIS
LIN {X 0.213,Y -617.107,Z 288.227,A 0.000,B 0.000,C 90.000,E1 256.881} C_DIS
LIN {X 0.033,Y -619.468,Z 288.219,A 0.000,B 0.000,C 90.000,E1 255.353} C_DIS
LIN {X -0.106,Y -620.978,Z 288.213,A 0.000,B 0.000,C 90.000,E1 254.338} C_DIS
LIN {X 0.001,Y -621.874,Z 288.209,A 0.000,B 0.000,C 90.000,E1 253.559} C_DIS
LIN {X -0.101,Y -622.711,Z 288.203,A 0.000,B 0.000,C 90.000,E1 252.543} C_DIS
LIN {X -0.221,Y -623.633,Z 288.196,A 0.000,B 0.000,C 90.000,E1 251.275} C_DIS
LIN {X -0.094,Y -623.950,Z 288.192,A 0.000,B 0.000,C 90.000,E1 250.496} C_DIS
LIN {X 0.237,Y -624.027,Z 288.186,A 0.000,B 0.000,C 90.000,E1 249.444} C_DIS
LIN {X -0.225,Y -623.817,Z 288.182,A 0.000,B 0.000,C 90.000,E1 248.720} C_DIS
LIN {X 0.109,Y -623.201,Z 288.176,A 0.000,B 0.000,C 90.000,E1 247.667} C_DIS
LIN {X -0.134,Y -622.749,Z 288.173,A 0.000,B 0.000,C 90.000,E1 247.177} C_DIS
LIN {X -0.136,Y -621.806,Z 288.169,A 0.000,B 0.000,C 90.000,E1 246.410} C_DIS
LIN {X 0.168,Y -620.300,Z 288.163,A 0.000,B 0.000,C 90.000,E1 245.357} C_DIS
LIN {X 0.143,Y -618.323,Z 288.158,A 0.000,B 0.000,C 90.000,E1 244.332} C_DIS
LIN {X -0.163,Y -616.599,Z 288.153,A 0.000,B 0.000,C 90.000,E1 243.589} C_DIS
LIN {X 0.043,Y -614.118,Z 288.147,A 0.000,B 0.000,C 90.000,E1 242.538} C_DIS
LIN {X -0.100,Y -610.732,Z 288.140,A 0.000,B 0.000,C 90.000,E1 241.257} C_DIS
LIN {X 0.234,Y -606.375,Z 288.132,A 0.000,B 0.000,C 90.000,E1 239.665} C_DIS
LIN {X -0.282,Y -602.600,Z 288.124,A 0.000,B 0.000,C 90.000,E1 238.408} C_DIS
LIN {X 0.280,Y -598.726,Z 288.117,A 0.000,B 0.000,C 90.000,E1 237.041} C_DIS
LIN {X -0.056,Y -594.657,Z 288.110,A 0.000,B 0.000,C 90.000,E1 235.754} C_DIS
LIN {X -0.005,Y -591.247,Z 288.104,A 0.000,B 0.000,C 90.000,E1 234.689} C_DIS
LIN {X 0.153,Y -583.462,Z 288.091,A 0.000,B 0.000,C 90.000,E1 232.271} C_DIS
LIN {X -0.074,Y -578.495,Z 288.082,A 0.000,B 0.000,C 90.000,E1 230.678} C_DIS
LIN {X -0.136,Y -570.827,Z 288.068,A 0.000,B 0.000,C 90.000,E1 228.243} C_DIS
LIN {X -0.009,Y -566.656,Z 288.060,A 0.000,B 0.000,C 90.000,E1 226.863} C_DIS
LIN {X -0.303,Y -561.545,Z 288.051,A 0.000,B 0.000,C 90.000,E1 225.243} C_DIS
LIN {X 0.091,Y -556.377,Z 288.042,A 0.000,B 0.000,C 90.000,E1 223.542} C_DIS
